LIN {X 0,Y 178.694,Z 336.057,A -85,B 0,C 180,E1 -23455.237,E2 -23455.237} C_VEL
LIN {X 0,Y 177.657,Z 345.122,A -85,B 0,C 180,E1 -23457.721,E2 -23457.721} C_VEL
LIN {X 0,Y 176.562,Z 350.916,A -85,B 0,C 180,E1 -23459.502,E2 -23459.502} C_VEL
LIN {X 0,Y 173.307,Z 359.118,A -85,B 0,C 180,E1 -23462.202,E2 -23462.202} C_VEL
LIN {X 0,Y 169.92,Z 367.179,A -85,B 0,C 180,E1 -23465.569,E2 -23465.569} C_VEL
LIN {X 0,Y 167.647,Z 372.655,A -85,B 0,C 180,E1 -23468.481,E2 -23468.481} C_VEL
LIN {X 0,Y 164.982,Z 378.808,A -85,B 0,C 180,E1 -23472.651,E2 -23472.651} C_VEL
LIN {X 0,Y 163.397,Z 382.822,A -85,B 0,C 180,E1 -23476.316,E2 -23476.316} C_VEL
LIN {X 0,Y 162.479,Z 385.804,A -85,B 0,C 180,E1 -23480.037,E2 -23480.037} C_VEL
LIN {X 0,Y 162.174,Z 387.231,A -85,B 0,C 180,E1 -23482.53,E2 -23482.53} C_VEL
LIN {X 0,Y 162.092,Z 388.497,A -85,B 0,C 180,E1 -23485.741,E2 -23485.741} C_VEL
LIN {X 0,Y 162.298,Z 389.115,A -85,B 0,C 180,E1 -23490,E2 -23490} C_VEL
LIN {X 0,Y 162.074,Z 388.506,A -85,B 0,C 180,E1 -23494.173,E2 -23494.173} C_VEL
LIN {X 0,Y 162.172,Z 387.205,A -85,B 0,C 180,E1 -23497.471,E2 -23497.471} C_VEL
LIN {X 0,Y 162.476,Z 385.767,A -85,B 0,C 180,E1 -23499.964,E2 -23499.964} C_VEL
LIN {X 0,Y 163.397,Z 382.767,A -85,B 0,C 180,E1 -23503.684,E2 -23503.684} C_VEL
LIN {X 0,Y 164.978,Z 378.732,A -85,B 0,C 180,E1 -23507.35,E2 -23507.35} C_VEL
LIN {X 0,Y 167.639,Z 372.55,A -85,B 0,C 180,E1 -23511.521,E2 -23511.521} C_VEL
LIN {X 0,Y 170.317,Z 366.243,A -85,B 0,C 180,E1 -23514.795,E2 -23514.795} C_VEL
LIN {X 0,Y 173.896,Z 357.578,A -85,B 0,C 180,E1 -23518.302,E2 -23518.302} C_VEL
LIN {X 0,Y 174.762,Z 353.72,A -85,B 0,C 180,E1 -23519.737,E2 -23519.737} C_VEL
LIN {X 0,Y 174.495,Z 349.857,A -85,B 0,C 180,E1 -23521.217,E2 -23521.217} C_VEL
LIN {X 0,Y 172.381,Z 339.088,A -85,B 0,C 180,E1 -23525.119,E2 -23525.119} C_VEL
LIN {X 0,Y 172.396,Z 336.052,A -85,B 0,C 180,E1 -23526.015,E2 -23526.015} C_VEL
LIN {X 0,Y 172.819,Z 325.215,A -85,B 0,C 180,E1 -23528.794,E2 -23528.794} C_VEL
LIN {X 0,Y 172.362,Z 314.414,A -85,B 0,C 180,E1 -23531.293,E2 -23531.293} C_VEL
LIN {X 0,Y 171.168,Z 305.853,A -85,B 0,C 180,E1 -23533.214,E2 -23533.214} C_VEL
LIN {X 0,Y 169.717,Z 301.249,A -85,B 0,C 180,E1 -23534.412,E2 -23534.412} C_VEL
LIN {X 0,Y 166.792,Z 294.609,A -85,B 0,C 180,E1 -23536.361,E2 -23536.361} C_VEL
LIN {X 0,Y 164.788,Z 290.322,A -85,B 0,C 180,E1 -23537.639,E2 -23537.639} C_VEL
LIN {X 0,Y 162.711,Z 286.562,A -85,B 0,C 180,E1 -23538.89,E2 -23538.89} C_VEL
LIN {X 0,Y 161.91,Z 284.961,A -85,B 0,C 180,E1 -23539.375,E2 -23539.375} C_VEL
LIN {X 0,Y 159.811,Z 281.715,A -85,B 0,C 180,E1 -23540.586,E2 -23540.586} C_VEL
LIN {X 0,Y 159.083,Z 279.423,A -85,B 0,C 180,E1 -23541.187,E2 -23541.187} C_VEL
LIN {X 0,Y 158.518,Z 275.963,A -85,B 0,C 180,E1 -23547.393,E2 -23547.393} C_VEL
LIN {X 0,Y 158.079,Z 272.941,A -85,B 0,C 180,E1 -23553.603,E2 -23553.603} C_VEL
LIN {X 0,Y 157.67,Z 270.525,A -85,B 0,C 180,E1 -23559.401,E2 -23559.401} C_VEL
LIN {X 0,Y 157.456,Z 268.872,A -85,B 0,C 180,E1 -23564.466,E2 -23564.466} C_VEL
LIN {X 0,Y 157.692,Z 268.842,A -85,B 0,C 180,E1 -23569.731,E2 -23569.731} C_VEL
LIN {X 0,Y 157.769,Z 268.832,A -85,B 0,C 180,E1 -23572.32,E2 -23572.32} C_VEL
LIN {X 0,Y 157.974,Z 268.806,A -85,B 0,C 180,E1 -23577.45,E2 -23577.45} C_VEL
LIN {X 0,Y 158.242,Z 268.772,A -85,B 0,C 180,E1 -23580,E2 -23580} C_VEL
LIN {X 0,Y 157.767,Z 268.833,A -85,B 0,C 180,E1 -23587.68,E2 -23587.68} C_VEL
LIN {X 0,Y 157.636,Z 268.847,A -85,B 0,C 180,E1 -23591.229,E2 -23591.229} C_VEL
LIN {X 0,Y 157.425,Z 268.874,A -85,B 0,C 180,E1 -23595.537,E2 -23595.537} C_VEL
LIN {X 0,Y 157.359,Z 268.881,A -85,B 0,C 180,E1 -23600.935,E2 -23600.935} C_VEL
LIN {X 0,Y 157.312,Z 268.888,A -85,B 0,C 180,E1 -23606.681,E2 -23606.681} C_VEL
LIN {X 0,Y 157.27,Z 268.895,A -85,B 0,C 180,E1 -23612.429,E2 -23612.429} C_VEL
LIN {X 0,Y 157.244,Z 268.897,A -85,B 0,C 180,E1 -23617.473,E2 -23617.473} C_VEL
LIN {X 0,Y 157.215,Z 268.901,A -85,B 0,C 180,E1 -23618.189,E2 -23618.189} C_VEL
LIN {X 0,Y 158.173,Z 271.614,A -85,B 0,C 180,E1 -23618.959,E2 -23618.959} C_VEL
LIN {X 0,Y 160.167,Z 273.789,A -85,B 0,C 180,E1 -23620.092,E2 -23620.092} C_VEL
LIN {X 0,Y 162.728,Z 277.922,A -85,B 0,C 180,E1 -23621.711,E2 -23621.711} C_VEL
LIN {X 0,Y 163.851,Z 279.647,A -85,B 0,C 180,E1 -23622.394,E2 -23622.394} C_VEL
LIN {X 0,Y 167.352,Z 285.536,A -85,B 0,C 180,E1 -23624.619,E2 -23624.619} C_VEL
LIN {X 0,Y 171.406,Z 294.402,A -85,B 0,C 180,E1 -23627.565,E2 -23627.565} C_VEL
LIN {X 0,Y 174.028,Z 302.719,A -85,B 0,C 180,E1 -23630.113,E2 -23630.113} C_VEL
LIN {X 0,Y 175.916,Z 312.518,A -85,B 0,C 180,E1 -23633.037,E2 -23633.037} C_VEL
LIN {X 0,Y 176.6,Z 320.843,A -85,B 0,C 180,E1 -23635.599,E2 -23635.599} C_VEL
LIN {X 0,Y 176.522,Z 323.692,A -85,B 0,C 180,E1 -23636.477,E2 -23636.477} C_VEL
LIN {X 0,Y 173.339,Z 332.499,A -85,B 0,C 180,E1 -23638.872,E2 -23638.872} C_VEL
LIN {X 0,Y 169.236,Z 342.093,A -85,B 0,C 180,E1 -23642.148,E2 -23642.148} C_VEL
LIN {X 0,Y 165.684,Z 349.73,A -85,B 0,C 180,E1 -23645.57,E2 -23645.57} C_VEL
LIN {X 0,Y 162.142,Z 356.74,A -85,B 0,C 180,E1 -23649.71,E2 -23649.71} C_VEL
LIN {X 0,Y 159.687,Z 361.404,A -85,B 0,C 180,E1 -23653.377,E2 -23653.377} C_VEL
LIN {X 0,Y 157.888,Z 364.961,A -85,B 0,C 180,E1 -23657.14,E2 -23657.14} C_VEL
LIN {X 0,Y 156.754,Z 367.275,A -85,B 0,C 180,E1 -23660.527,E2 -23660.527} C_VEL
LIN {X 0,Y 155.826,Z 369.151,A -85,B 0,C 180,E1 -23664.824,E2 -23664.824} C_VEL
LIN {X 0,Y 155.406,Z 369.98,A -85,B 0,C 180,E1 -23670,E2 -23670} C_VEL
LIN {X 0,Y 155.513,Z 369.784,A -85,B 0,C 180,E1 -23672.59,E2 -23672.59} C_VEL
LIN {X 0,Y 155.814,Z 369.201,A -85,B 0,C 180,E1 -23675.175,E2 -23675.175} C_VEL
LIN {X 0,Y 156.942,Z 366.896,A -85,B 0,C 180,E1 -23680.318,E2 -23680.318} C_VEL
LIN {X 0,Y 158.396,Z 364.048,A -85,B 0,C 180,E1 -23684.124,E2 -23684.124} C_VEL
LIN {X 0,Y 160.389,Z 360.182,A -85,B 0,C 180,E1 -23687.862,E2 -23687.862} C_VEL
LIN {X 0,Y 162.993,Z 355.185,A -85,B 0,C 180,E1 -23691.5,E2 -23691.5} C_VEL
LIN {X 0,Y 166.103,Z 348.887,A -85,B 0,C 180,E1 -23695.031,E2 -23695.031} C_VEL
LIN {X 0,Y 169.836,Z 340.996,A -85,B 0,C 180,E1 -23698.417,E2 -23698.417} C_VEL
LIN {X 0,Y 173.294,Z 332.948,A -85,B 0,C 180,E1 -23701.137,E2 -23701.137} C_VEL
LIN {X 0,Y 176.772,Z 323.142,A -85,B 0,C 180,E1 -23703.821,E2 -23703.821} C_VEL
LIN {X 0,Y 176.286,Z 315.562,A -85,B 0,C 180,E1 -23706.21,E2 -23706.21} C_VEL
LIN {X 0,Y 174.842,Z 306.158,A -85,B 0,C 180,E1 -23709.041,E2 -23709.041} C_VEL
LIN {X 0,Y 172.954,Z 298.802,A -85,B 0,C 180,E1 -23711.256,E2 -23711.256} C_VEL
LIN {X 0,Y 169.65,Z 290.247,A -85,B 0,C 180,E1 -23713.981,E2 -23713.981} C_VEL
LIN {X 0,Y 165.677,Z 282.509,A -85,B 0,C 180,E1 -23716.682,E2 -23716.682} C_VEL
LIN {X 0,Y 162.745,Z 277.931,A -85,B 0,C 180,E1 -23718.501,E2 -23718.501} C_VEL
LIN {X 0,Y 160.785,Z 274.801,A -85,B 0,C 180,E1 -23719.739,E2 -23719.739} C_VEL
LIN {X 0,Y 160.185,Z 273.812,A -85,B 0,C 180,E1 -23720.126,E2 -23720.126} C_VEL
LIN {X 0,Y 158.103,Z 271.534,A -85,B 0,C 180,E1 -23721.317,E2 -23721.317} C_VEL
LIN {X 0,Y 157.207,Z 268.903,A -85,B 0,C 180,E1 -23722.045,E2 -23722.045} C_VEL
LIN {X 0,Y 157.279,Z 268.894,A -85,B 0,C 180,E1 -23724.486,E2 -23724.486} C_VEL
LIN {X 0,Y 157.284,Z 268.89,A -85,B 0,C 180,E1 -23728.102,E2 -23728.102} C_VEL
LIN {X 0,Y 157.31,Z 268.889,A -85,B 0,C 180,E1 -23733.464,E2 -23733.464} C_VEL
LIN {X 0,Y 157.378,Z 268.882,A -85,B 0,C 180,E1 -23739.684,E2 -23739.684} C_VEL
LIN {X 0,Y 157.426,Z 268.873,A -85,B 0,C 180,E1 -23744.463,E2 -23744.463} C_VEL
LIN {X 0,Y 157.748,Z 268.831,A -85,B 0,C 180,E1 -23749.734,E2 -23749.734} C_VEL
LIN {X 0,Y 157.82,Z 268.822,A -85,B 0,C 180,E1 -23752.322,E2 -23752.322} C_VEL
LIN {X 0,Y 158.241,Z 268.769,A -85,B 0,C 180,E1 -23760,E2 -23760} C_VEL
LIN {X 0,Y 157.714,Z 268.841,A -85,B 0,C 180,E1 -23765.113,E2 -23765.113} C_VEL
LIN {X 0,Y 157.768,Z 268.833,A -85,B 0,C 180,E1 -23767.68,E2 -23767.68} C_VEL
LIN {X 0,Y 157.659,Z 268.847,A -85,B 0,C 180,E1 -23771.275,E2 -23771.275} C_VEL
LIN {X 0,Y 157.443,Z 268.869,A -85,B 0,C 180,E1 -23775.535,E2 -23775.535} C_VEL
LIN {X 0,Y 157.696,Z 270.702,A -85,B 0,C 180,E1 -23780.887,E2 -23780.887} C_VEL
LIN {X 0,Y 158.056,Z 273.015,A -85,B 0,C 180,E1 -23786.401,E2 -23786.401} C_VEL
LIN {X 0,Y 158.487,Z 276.059,A -85,B 0,C 180,E1 -23792.59,E2 -23792.59} C_VEL
LIN {X 0,Y 159.068,Z 279.471,A -85,B 0,C 180,E1 -23798.716,E2 -23798.716} C_VEL
LIN {X 0,Y 160.384,Z 282.857,A -85,B 0,C 180,E1 -23799.652,E2 -23799.652} C_VEL
LIN {X 0,Y 162.485,Z 285.847,A -85,B 0,C 180,E1 -23800.826,E2 -23800.826} C_VEL
LIN {X 0,Y 164.332,Z 289.647,A -85,B 0,C 180,E1 -23801.994,E2 -23801.994} C_VEL
LIN {X 0,Y 165.621,Z 292.033,A -85,B 0,C 180,E1 -23802.762,E2 -23802.762} C_VEL
LIN {X 0,Y 169.159,Z 299.71,A -85,B 0,C 180,E1 -23805.066,E2 -23805.066} C_VEL
LIN {X 0,Y 171.197,Z 305.8,A -85,B 0,C 180,E1 -23806.69,E2 -23806.69} C_VEL
LIN {X 0,Y 172.473,Z 314.952,A -85,B 0,C 180,E1 -23808.755,E2 -23808.755} C_VEL
LIN {X 0,Y 172.901,Z 325.446,A -85,B 0,C 180,E1 -23811.2,E2 -23811.2} C_VEL
LIN {X 0,Y 172.449,Z 336.06,A -85,B 0,C 180,E1 -23813.921,E2 -23813.921} C_VEL
LIN {X 0,Y 171.405,Z 344.677,A -85,B 0,C 180,E1 -23816.391,E2 -23816.391} C_VEL
LIN {X 0,Y 169.797,Z 352.288,A -85,B 0,C 180,E1 -23818.843,E2 -23818.843} C_VEL
LIN {X 0,Y 165.739,Z 361.567,A -85,B 0,C 180,E1 -23822.196,E2 -23822.196} C_VEL
LIN {X 0,Y 162.419,Z 369.198,A -85,B 0,C 180,E1 -23825.816,E2 -23825.816} C_VEL
LIN {X 0,Y 159.707,Z 375.066,A -85,B 0,C 180,E1 -23829.388,E2 -23829.388} C_VEL
LIN {X 0,Y 157.535,Z 379.828,A -85,B 0,C 180,E1 -23833.143,E2 -23833.143} C_VEL
LIN {X 0,Y 156.082,Z 383.483,A -85,B 0,C 180,E1 -23836.989,E2 -23836.989} C_VEL
LIN {X 0,Y 155.464,Z 385.375,A -85,B 0,C 180,E1 -23839.582,E2 -23839.582} C_VEL
LIN {X 0,Y 155.011,Z 387.829,A -85,B 0,C 180,E1 -23844.798,E2 -23844.798} C_VEL
LIN {X 0,Y 155.026,Z 388.459,A -85,B 0,C 180,E1 -23847.402,E2 -23847.402} C_VEL
LIN {X 0,Y 155.214,Z 388.689,A -85,B 0,C 180,E1 -23850,E2 -23850} C_VEL
LIN {X 0,Y 155.002,Z 388.164,A -85,B 0,C 180,E1 -23854.045,E2 -23854.045} C_VEL
LIN {X 0,Y 155.111,Z 386.776,A -85,B 0,C 180,E1 -23857.813,E2 -23857.813} C_VEL
LIN {X 0,Y 155.462,Z 385.337,A -85,B 0,C 180,E1 -23860.418,E2 -23860.418} C_VEL
LIN {X 0,Y 156.468,Z 382.336,A -85,B 0,C 180,E1 -23864.303,E2 -23864.303} C_VEL
LIN {X 0,Y 158.195,Z 378.302,A -85,B 0,C 180,E1 -23868.119,E2 -23868.119} C_VEL
LIN {X 0,Y 161.045,Z 372.12,A -85,B 0,C 180,E1 -23872.449,E2 -23872.449} C_VEL
LIN {X 0,Y 163.99,Z 365.503,A -85,B 0,C 180,E1 -23875.989,E2 -23875.989} C_VEL
LIN {X 0,Y 167.695,Z 357.031,A -85,B 0,C 180,E1 -23879.501,E2 -23879.501} C_VEL
LIN {X 0,Y 169.785,Z 352.093,A -85,B 0,C 180,E1 -23881.16,E2 -23881.16} C_VEL
LIN {X 0,Y 171.535,Z 343.379,A -85,B 0,C 180,E1 -23883.934,E2 -23883.934} C_VEL
LIN {X 0,Y 172.396,Z 336.052,A -85,B 0,C 180,E1 -23886.015,E2 -23886.015} C_VEL
LIN {X 0,Y 172.137,Z 331.689,A -85,B 0,C 180,E1 -23887.336,E2 -23887.336} C_VEL
LIN {X 0,Y 170.969,Z 327.609,A -85,B 0,C 180,E1 -23888.729,E2 -23888.729} C_VEL
LIN {X 0,Y 167.747,Z 319.532,A -85,B 0,C 180,E1 -23891.534,E2 -23891.534} C_VEL
LIN {X 0,Y 166.552,Z 315.06,A -85,B 0,C 180,E1 -23892.841,E2 -23892.841} C_VEL
LIN {X 0,Y 166.322,Z 313.452,A -85,B 0,C 180,E1 -23893.241,E2 -23893.241} C_VEL
LIN {X 0,Y 165.249,Z 307.101,A -85,B 0,C 180,E1 -23894.848,E2 -23894.848} C_VEL
LIN {X 0,Y 161.779,Z 298.409,A -85,B 0,C 180,E1 -23897.606,E2 -23897.606} C_VEL
LIN {X 0,Y 160.213,Z 294.941,A -85,B 0,C 180,E1 -23898.744,E2 -23898.744} C_VEL
LIN {X 0,Y 157.631,Z 289.802,A -85,B 0,C 180,E1 -23900.555,E2 -23900.555} C_VEL
LIN {X 0,Y 155.501,Z 285.739,A -85,B 0,C 180,E1 -23902.049,E2 -23902.049} C_VEL
LIN {X 0,Y 154.729,Z 284.47,A -85,B 0,C 180,E1 -23902.555,E2 -23902.555} C_VEL
LIN {X 0,Y 152.517,Z 281.225,A -85,B 0,C 180,E1 -23904.019,E2 -23904.019} C_VEL
LIN {X 0,Y 151.752,Z 278.759,A -85,B 0,C 180,E1 -23904.728,E2 -23904.728} C_VEL
LIN {X 0,Y 151.369,Z 276.46,A -85,B 0,C 180,E1 -23909.288,E2 -23909.288} C_VEL
LIN {X 0,Y 151.205,Z 275.058,A -85,B 0,C 180,E1 -23912.303,E2 -23912.303} C_VEL
LIN {X 0,Y 150.771,Z 272.37,A -85,B 0,C 180,E1 -23918.794,E2 -23918.794} C_VEL
LIN {X 0,Y 150.54,Z 270.645,A -85,B 0,C 180,E1 -23923.733,E2 -23923.733} C_VEL
LIN {X 0,Y 150.445,Z 269.8,A -85,B 0,C 180,E1 -23926.493,E2 -23926.493} C_VEL
LIN {X 0,Y 150.626,Z 269.724,A -85,B 0,C 180,E1 -23929.244,E2 -23929.244} C_VEL
LIN {X 0,Y 150.707,Z 269.713,A -85,B 0,C 180,E1 -23931.958,E2 -23931.958} C_VEL
LIN {X 0,Y 151.204,Z 269.649,A -85,B 0,C 180,E1 -23940,E2 -23940} C_VEL
LIN {X 0,Y 150.705,Z 269.712,A -85,B 0,C 180,E1 -23948.042,E2 -23948.042} C_VEL
LIN {X 0,Y 150.578,Z 269.726,A -85,B 0,C 180,E1 -23951.433,E2 -23951.433} C_VEL
LIN {X 0,Y 150.333,Z 269.759,A -85,B 0,C 180,E1 -23956.29,E2 -23956.29} C_VEL
LIN {X 0,Y 150.342,Z 269.755,A -85,B 0,C 180,E1 -23960.78,E2 -23960.78} C_VEL
LIN {X 0,Y 150.241,Z 269.771,A -85,B 0,C 180,E1 -23967.277,E2 -23967.277} C_VEL
LIN {X 0,Y 150.211,Z 269.773,A -85,B 0,C 180,E1 -23972.628,E2 -23972.628} C_VEL
LIN {X 0,Y 150.188,Z 269.775,A -85,B 0,C 180,E1 -23974.67,E2 -23974.67} C_VEL
LIN {X 0,Y 151.132,Z 272.438,A -85,B 0,C 180,E1 -23975.541,E2 -23975.541} C_VEL
LIN {X 0,Y 153.125,Z 274.667,A -85,B 0,C 180,E1 -23976.874,E2 -23976.874} C_VEL
LIN {X 0,Y 153.818,Z 275.484,A -85,B 0,C 180,E1 -23977.344,E2 -23977.344} C_VEL
LIN {X 0,Y 155.642,Z 278.625,A -85,B 0,C 180,E1 -23978.697,E2 -23978.697} C_VEL
LIN {X 0,Y 157.036,Z 280.466,A -85,B 0,C 180,E1 -23979.624,E2 -23979.624} C_VEL
LIN {X 0,Y 160.948,Z 287.028,A -85,B 0,C 180,E1 -23982.427,E2 -23982.427} C_VEL
LIN {X 0,Y 164.358,Z 293.877,A -85,B 0,C 180,E1 -23985.052,E2 -23985.052} C_VEL
LIN {X 0,Y 166.932,Z 300.819,A -85,B 0,C 180,E1 -23987.459,E2 -23987.459} C_VEL
LIN {X 0,Y 168.746,Z 307.844,A -85,B 0,C 180,E1 -23989.763,E2 -23989.763} C_VEL
LIN {X 0,Y 170.042,Z 316.864,A -85,B 0,C 180,E1 -23992.67,E2 -23992.67} C_VEL
LIN {X 0,Y 170.378,Z 324.858,A -85,B 0,C 180,E1 -23995.347,E2 -23995.347} C_VEL
LIN {X 0,Y 166.591,Z 334.695,A -85,B 0,C 180,E1 -23998.173,E2 -23998.173} C_VEL
LIN {X 0,Y 163.016,Z 342.522,A -85,B 0,C 180,E1 -24000.986,E2 -24000.986} C_VEL
LIN {X 0,Y 159.26,Z 350.158,A -85,B 0,C 180,E1 -24004.516,E2 -24004.516} C_VEL
LIN {X 0,Y 155.519,Z 357.169,A -85,B 0,C 180,E1 -24008.806,E2 -24008.806} C_VEL
LIN {X 0,Y 152.912,Z 361.832,A -85,B 0,C 180,E1 -24012.617,E2 -24012.617} C_VEL
LIN {X 0,Y 150.973,Z 365.389,A -85,B 0,C 180,E1 -24016.54,E2 -24016.54} C_VEL
LIN {X 0,Y 149.684,Z 367.872,A -85,B 0,C 180,E1 -24020.402,E2 -24020.402} C_VEL
LIN {X 0,Y 148.776,Z 369.578,A -85,B 0,C 180,E1 -24024.578,E2 -24024.578} C_VEL
LIN {X 0,Y 148.347,Z 370.405,A -85,B 0,C 180,E1 -24030,E2 -24030} C_VEL
LIN {X 0,Y 148.439,Z 370.21,A -85,B 0,C 180,E1 -24032.713,E2 -24032.713} C_VEL
LIN {X 0,Y 148.763,Z 369.627,A -85,B 0,C 180,E1 -24035.421,E2 -24035.421} C_VEL
LIN {X 0,Y 149.982,Z 367.322,A -85,B 0,C 180,E1 -24040.803,E2 -24040.803} C_VEL
LIN {X 0,Y 151.534,Z 364.474,A -85,B 0,C 180,E1 -24044.778,E2 -24044.778} C_VEL
LIN {X 0,Y 153.649,Z 360.608,A -85,B 0,C 180,E1 -24048.674,E2 -24048.674} C_VEL
LIN {X 0,Y 156.419,Z 355.61,A -85,B 0,C 180,E1 -24052.452,E2 -24052.452} C_VEL
LIN {X 0,Y 159.703,Z 349.312,A -85,B 0,C 180,E1 -24056.108,E2 -24056.108} C_VEL
LIN {X 0,Y 163.643,Z 341.42,A -85,B 0,C 180,E1 -24059.597,E2 -24059.597} C_VEL
LIN {X 0,Y 167.265,Z 333.372,A -85,B 0,C 180,E1 -24062.392,E2 -24062.392} C_VEL
LIN {X 0,Y 170.487,Z 324.68,A -85,B 0,C 180,E1 -24064.87,E2 -24064.87} C_VEL
LIN {X 0,Y 170.066,Z 316.091,A -85,B 0,C 180,E1 -24067.741,E2 -24067.741} C_VEL
LIN {X 0,Y 168.502,Z 306.306,A -85,B 0,C 180,E1 -24070.9,E2 -24070.9} C_VEL
LIN {X 0,Y 165.814,Z 297.331,A -85,B 0,C 180,E1 -24073.9,E2 -24073.9} C_VEL
LIN {X 0,Y 162.05,Z 288.967,A -85,B 0,C 180,E1 -24077.001,E2 -24077.001} C_VEL
LIN {X 0,Y 158.675,Z 283.229,A -85,B 0,C 180,E1 -24079.418,E2 -24079.418} C_VEL
LIN {X 0,Y 156.462,Z 279.471,A -85,B 0,C 180,E1 -24081.034,E2 -24081.034} C_VEL
LIN {X 0,Y 154.281,Z 276.557,A -85,B 0,C 180,E1 -24082.509,E2 -24082.509} C_VEL
LIN {X 0,Y 153.407,Z 274.854,A -85,B 0,C 180,E1 -24083.206,E2 -24083.206} C_VEL
LIN {X 0,Y 151.282,Z 272.7,A -85,B 0,C 180,E1 -24084.602,E2 -24084.602} C_VEL
LIN {X 0,Y 150.285,Z 270.385,A -85,B 0,C 180,E1 -24085.457,E2 -24085.457} C_VEL
LIN {X 0,Y 150.195,Z 269.774,A -85,B 0,C 180,E1 -24085.637,E2 -24085.637} C_VEL
LIN {X 0,Y 150.192,Z 269.773,A -85,B 0,C 180,E1 -24089.02,E2 -24089.02} C_VEL
LIN {X 0,Y 150.239,Z 269.771,A -85,B 0,C 180,E1 -24092.722,E2 -24092.722} C_VEL
LIN {X 0,Y 150.34,Z 269.756,A -85,B 0,C 180,E1 -24099.22,E2 -24099.22} C_VEL
LIN {X 0,Y 150.333,Z 269.759,A -85,B 0,C 180,E1 -24103.71,E2 -24103.71} C_VEL
LIN {X 0,Y 150.662,Z 269.713,A -85,B 0,C 180,E1 -24109.246,E2 -24109.246} C_VEL
LIN {X 0,Y 150.756,Z 269.703,A -85,B 0,C 180,E1 -24111.96,E2 -24111.96} C_VEL
LIN {X 0,Y 151.203,Z 269.646,A -85,B 0,C 180,E1 -24120,E2 -24120} C_VEL
LIN {X 0,Y 150.705,Z 269.714,A -85,B 0,C 180,E1 -24128.042,E2 -24128.042} C_VEL
LIN {X 0,Y 150.591,Z 269.726,A -85,B 0,C 180,E1 -24131.461,E2 -24131.461} C_VEL
LIN {X 0,Y 150.448,Z 269.87,A -85,B 0,C 180,E1 -24133.507,E2 -24133.507} C_VEL
LIN {X 0,Y 150.684,Z 271.655,A -85,B 0,C 180,E1 -24139.055,E2 -24139.055} C_VEL
LIN {X 0,Y 150.952,Z 273.87,A -85,B 0,C 180,E1 -24144.773,E2 -24144.773} C_VEL
LIN {X 0,Y 151.183,Z 275.265,A -85,B 0,C 180,E1 -24147.964,E2 -24147.964} C_VEL
LIN {X 0,Y 151.585,Z 278.099,A -85,B 0,C 180,E1 -24153.804,E2 -24153.804} C_VEL
LIN {X 0,Y 151.745,Z 278.823,A -85,B 0,C 180,E1 -24155.172,E2 -24155.172} C_VEL
LIN {X 0,Y 152.756,Z 281.769,A -85,B 0,C 180,E1 -24156.018,E2 -24156.018} C_VEL
LIN {X 0,Y 155.488,Z 285.652,A -85,B 0,C 180,E1 -24157.796,E2 -24157.796} C_VEL
LIN {X 0,Y 157.33,Z 289.336,A -85,B 0,C 180,E1 -24159.122,E2 -24159.122} C_VEL
LIN {X 0,Y 158.516,Z 291.379,A -85,B 0,C 180,E1 -24159.903,E2 -24159.903} C_VEL
LIN {X 0,Y 161.197,Z 296.995,A -85,B 0,C 180,E1 -24161.831,E2 -24161.831} C_VEL
LIN {X 0,Y 164.503,Z 304.814,A -85,B 0,C 180,E1 -24164.369,E2 -24164.369} C_VEL
LIN {X 0,Y 166.074,Z 310.645,A -85,B 0,C 180,E1 -24166.006,E2 -24166.006} C_VEL
LIN {X 0,Y 166.793,Z 320.116,A -85,B 0,C 180,E1 -24168.292,E2 -24168.292} C_VEL
LIN {X 0,Y 166.747,Z 329.849,A -85,B 0,C 180,E1 -24170.786,E2 -24170.786} C_VEL
LIN {X 0,Y 165.899,Z 339.888,A -85,B 0,C 180,E1 -24173.624,E2 -24173.624} C_VEL
LIN {X 0,Y 164.496,Z 348.209,A -85,B 0,C 180,E1 -24176.261,E2 -24176.261} C_VEL
LIN {X 0,Y 163.019,Z 353.542,A -85,B 0,C 180,E1 -24178.122,E2 -24178.122} C_VEL
LIN {X 0,Y 158.812,Z 362.507,A -85,B 0,C 180,E1 -24181.594,E2 -24181.594} C_VEL
LIN {X 0,Y 155.567,Z 369.55,A -85,B 0,C 180,E1 -24185.172,E2 -24185.172} C_VEL
LIN {X 0,Y 153.026,Z 374.636,A -85,B 0,C 180,E1 -24188.444,E2 -24188.444} C_VEL
LIN {X 0,Y 150.71,Z 379.399,A -85,B 0,C 180,E1 -24192.356,E2 -24192.356} C_VEL
LIN {X 0,Y 149.123,Z 383.053,A -85,B 0,C 180,E1 -24196.371,E2 -24196.371} C_VEL
LIN {X 0,Y 148.469,Z 384.947,A -85,B 0,C 180,E1 -24199.086,E2 -24199.086} C_VEL
LIN {X 0,Y 147.929,Z 387.401,A -85,B 0,C 180,E1 -24204.548,E2 -24204.548} C_VEL
LIN {X 0,Y 147.933,Z 388.031,A -85,B 0,C 180,E1 -24207.277,E2 -24207.277} C_VEL
LIN {X 0,Y 148.13,Z 388.262,A -85,B 0,C 180,E1 -24210,E2 -24210} C_VEL
LIN {X 0,Y 147.94,Z 387.793,A -85,B 0,C 180,E1 -24213.95,E2 -24213.95} C_VEL
LIN {X 0,Y 148.044,Z 386.346,A -85,B 0,C 180,E1 -24218.188,E2 -24218.188} C_VEL
LIN {X 0,Y 148.467,Z 384.907,A -85,B 0,C 180,E1 -24220.915,E2 -24220.915} C_VEL
LIN {X 0,Y 149.566,Z 381.906,A -85,B 0,C 180,E1 -24224.978,E2 -24224.978} C_VEL
LIN {X 0,Y 151.416,Z 377.87,A -85,B 0,C 180,E1 -24228.96,E2 -24228.96} C_VEL
LIN {X 0,Y 154.499,Z 371.69,A -85,B 0,C 180,E1 -24233.456,E2 -24233.456} C_VEL
LIN {X 0,Y 157.664,Z 364.945,A -85,B 0,C 180,E1 -24237.188,E2 -24237.188} C_VEL
LIN {X 0,Y 161.54,Z 356.6,A -85,B 0,C 180,E1 -24240.744,E2 -24240.744} C_VEL
LIN {X 0,Y 163.566,Z 351.649,A -85,B 0,C 180,E1 -24242.486,E2 -24242.486} C_VEL
LIN {X 0,Y 165.393,Z 342.872,A -85,B 0,C 180,E1 -24245.397,E2 -24245.397} C_VEL
LIN {X 0,Y 166.436,Z 333.537,A -85,B 0,C 180,E1 -24248.139,E2 -24248.139} C_VEL
LIN {X 0,Y 166.816,Z 322.544,A -85,B 0,C 180,E1 -24251.011,E2 -24251.011} C_VEL
LIN {X 0,Y 166.322,Z 313.452,A -85,B 0,C 180,E1 -24253.241,E2 -24253.241} C_VEL
LIN {X 0,Y 165.664,Z 310.424,A -85,B 0,C 180,E1 -24254.069,E2 -24254.069} C_VEL
LIN {X 0,Y 164.464,Z 307.771,A -85,B 0,C 180,E1 -24254.985,E2 -24254.985} C_VEL
LIN {X 0,Y 161.161,Z 303.358,A -85,B 0,C 180,E1 -24256.995,E2 -24256.995} C_VEL
LIN {X 0,Y 153.729,Z 295.243,A -85,B 0,C 180,E1 -24261.424,E2 -24261.424} C_VEL
LIN {X 0,Y 151.603,Z 290.966,A -85,B 0,C 180,E1 -24263.148,E2 -24263.148} C_VEL
LIN {X 0,Y 148.668,Z 285.889,A -85,B 0,C 180,E1 -24265.439,E2 -24265.439} C_VEL
LIN {X 0,Y 147.872,Z 284.147,A -85,B 0,C 180,E1 -24266.123,E2 -24266.123} C_VEL
LIN {X 0,Y 145.349,Z 280.732,A -85,B 0,C 180,E1 -24268.072,E2 -24268.072} C_VEL
LIN {X 0,Y 144.432,Z 278.009,A -85,B 0,C 180,E1 -24269.072,E2 -24269.072} C_VEL
LIN {X 0,Y 144.083,Z 275.856,A -85,B 0,C 180,E1 -24273.96,E2 -24273.96} C_VEL
LIN {X 0,Y 143.776,Z 273.541,A -85,B 0,C 180,E1 -24279.991,E2 -24279.991} C_VEL
LIN {X 0,Y 143.554,Z 271.697,A -85,B 0,C 180,E1 -24285.831,E2 -24285.831} C_VEL
LIN {X 0,Y 143.597,Z 270.883,A -85,B 0,C 180,E1 -24288.71,E2 -24288.71} C_VEL
LIN {X 0,Y 143.63,Z 270.596,A -85,B 0,C 180,E1 -24291.559,E2 -24291.559} C_VEL
LIN {X 0,Y 144.164,Z 270.526,A -85,B 0,C 180,E1 -24300,E2 -24300} C_VEL
LIN {X 0,Y 143.627,Z 270.592,A -85,B 0,C 180,E1 -24308.442,E2 -24308.442} C_VEL
LIN {X 0,Y 143.504,Z 270.606,A -85,B 0,C 180,E1 -24311.621,E2 -24311.621} C_VEL
LIN {X 0,Y 143.272,Z 270.636,A -85,B 0,C 180,E1 -24317.117,E2 -24317.117} C_VEL
LIN {X 0,Y 143.269,Z 270.637,A -85,B 0,C 180,E1 -24321.244,E2 -24321.244} C_VEL
LIN {X 0,Y 143.185,Z 270.648,A -85,B 0,C 180,E1 -24327.931,E2 -24327.931} C_VEL
LIN {X 0,Y 143.168,Z 270.851,A -85,B 0,C 180,E1 -24330.413,E2 -24330.413} C_VEL
LIN {X 0,Y 144.077,Z 273.378,A -85,B 0,C 180,E1 -24331.422,E2 -24331.422} C_VEL
LIN {X 0,Y 146.25,Z 275.679,A -85,B 0,C 180,E1 -24333.159,E2 -24333.159} C_VEL
LIN {X 0,Y 147.004,Z 276.3,A -85,B 0,C 180,E1 -24333.725,E2 -24333.725} C_VEL
LIN {X 0,Y 148.731,Z 279.486,A -85,B 0,C 180,E1 -24335.266,E2 -24335.266} C_VEL
LIN {X 0,Y 150.329,Z 281.442,A -85,B 0,C 180,E1 -24336.485,E2 -24336.485} C_VEL
LIN {X 0,Y 154.983,Z 289.096,A -85,B 0,C 180,E1 -24340.256,E2 -24340.256} C_VEL
LIN {X 0,Y 157.922,Z 294.771,A -85,B 0,C 180,E1 -24342.74,E2 -24342.74} C_VEL
LIN {X 0,Y 160.864,Z 302.141,A -85,B 0,C 180,E1 -24345.65,E2 -24345.65} C_VEL
LIN {X 0,Y 163.002,Z 310.677,A -85,B 0,C 180,E1 -24348.694,E2 -24348.694} C_VEL
LIN {X 0,Y 164.026,Z 319.692,A -85,B 0,C 180,E1 -24351.815,E2 -24351.815} C_VEL
LIN {X 0,Y 164.195,Z 325.419,A -85,B 0,C 180,E1 -24353.878,E2 -24353.878} C_VEL
LIN {X 0,Y 163.868,Z 327.319,A -85,B 0,C 180,E1 -24354.485,E2 -24354.485} C_VEL
LIN {X 0,Y 159.848,Z 336.804,A -85,B 0,C 180,E1 -24357.411,E2 -24357.411} C_VEL
LIN {X 0,Y 155.479,Z 345.669,A -85,B 0,C 180,E1 -24360.926,E2 -24360.926} C_VEL
LIN {X 0,Y 151.707,Z 352.794,A -85,B 0,C 180,E1 -24364.626,E2 -24364.626} C_VEL
LIN {X 0,Y 148.944,Z 357.596,A -85,B 0,C 180,E1 -24367.822,E2 -24367.822} C_VEL
LIN {X 0,Y 146.175,Z 362.259,A -85,B 0,C 180,E1 -24371.789,E2 -24371.789} C_VEL
LIN {X 0,Y 144.097,Z 365.817,A -85,B 0,C 180,E1 -24375.885,E2 -24375.885} C_VEL
LIN {X 0,Y 142.563,Z 368.534,A -85,B 0,C 180,E1 -24380.387,E2 -24380.387} C_VEL
LIN {X 0,Y 141.731,Z 370.005,A -85,B 0,C 180,E1 -24384.308,E2 -24384.308} C_VEL
LIN {X 0,Y 141.265,Z 370.832,A -85,B 0,C 180,E1 -24390,E2 -24390} C_VEL
LIN {X 0,Y 141.367,Z 370.637,A -85,B 0,C 180,E1 -24392.849,E2 -24392.849} C_VEL
LIN {X 0,Y 141.717,Z 370.053,A -85,B 0,C 180,E1 -24395.692,E2 -24395.692} C_VEL
LIN {X 0,Y 142.456,Z 368.752,A -85,B 0,C 180,E1 -24399.355,E2 -24399.355} C_VEL
LIN {X 0,Y 144.084,Z 365.945,A -85,B 0,C 180,E1 -24404.116,E2 -24404.116} C_VEL
LIN {X 0,Y 146.142,Z 362.436,A -85,B 0,C 180,E1 -24408.215,E2 -24408.215} C_VEL
LIN {X 0,Y 148.878,Z 357.823,A -85,B 0,C 180,E1 -24412.188,E2 -24412.188} C_VEL
LIN {X 0,Y 152.776,Z 350.866,A -85,B 0,C 180,E1 -24416.648,E2 -24416.648} C_VEL
LIN {X 0,Y 156.809,Z 343.31,A -85,B 0,C 180,E1 -24420.279,E2 -24420.279} C_VEL
LIN {X 0,Y 160.565,Z 335.561,A -85,B 0,C 180,E1 -24423.17,E2 -24423.17} C_VEL
LIN {X 0,Y 164.259,Z 326.324,A -85,B 0,C 180,E1 -24425.961,E2 -24425.961} C_VEL
LIN {X 0,Y 163.974,Z 317.751,A -85,B 0,C 180,E1 -24429.027,E2 -24429.027} C_VEL
LIN {X 0,Y 162.642,Z 308.715,A -85,B 0,C 180,E1 -24432.182,E2 -24432.182} C_VEL
LIN {X 0,Y 160.118,Z 299.983,A -85,B 0,C 180,E1 -24435.389,E2 -24435.389} C_VEL
LIN {X 0,Y 157.391,Z 293.646,A -85,B 0,C 180,E1 -24437.948,E2 -24437.948} C_VEL
LIN {X 0,Y 154.398,Z 288.294,A -85,B 0,C 180,E1 -24440.412,E2 -24440.412} C_VEL
LIN {X 0,Y 152.116,Z 284.438,A -85,B 0,C 180,E1 -24442.284,E2 -24442.284} C_VEL
LIN {X 0,Y 149.715,Z 280.528,A -85,B 0,C 180,E1 -24444.278,E2 -24444.278} C_VEL
LIN {X 0,Y 147.528,Z 277.559,A -85,B 0,C 180,E1 -24446.02,E2 -24446.02} C_VEL
LIN {X 0,Y 146.699,Z 275.938,A -85,B 0,C 180,E1 -24446.801,E2 -24446.801} C_VEL
LIN {X 0,Y 144.423,Z 273.922,A -85,B 0,C 180,E1 -24448.56,E2 -24448.56} C_VEL
LIN {X 0,Y 143.21,Z 271.242,A -85,B 0,C 180,E1 -24449.8,E2 -24449.8} C_VEL
LIN {X 0,Y 143.107,Z 270.66,A -85,B 0,C 180,E1 -24449.979,E2 -24449.979} C_VEL
LIN {X 0,Y 143.151,Z 270.651,A -85,B 0,C 180,E1 -24453.777,E2 -24453.777} C_VEL
LIN {X 0,Y 143.285,Z 270.638,A -85,B 0,C 180,E1 -24459.919,E2 -24459.919} C_VEL
LIN {X 0,Y 143.35,Z 270.623,A -85,B 0,C 180,E1 -24465.81,E2 -24465.81} C_VEL
LIN {X 0,Y 143.595,Z 270.593,A -85,B 0,C 180,E1 -24468.71,E2 -24468.71} C_VEL
LIN {X 0,Y 143.675,Z 270.587,A -85,B 0,C 180,E1 -24471.561,E2 -24471.561} C_VEL
LIN {X 0,Y 144.163,Z 270.522,A -85,B 0,C 180,E1 -24480,E2 -24480} C_VEL
LIN {X 0,Y 143.629,Z 270.593,A -85,B 0,C 180,E1 -24488.441,E2 -24488.441} C_VEL
LIN {X 0,Y 143.589,Z 271.097,A -85,B 0,C 180,E1 -24491.789,E2 -24491.789} C_VEL
LIN {X 0,Y 143.657,Z 272.657,A -85,B 0,C 180,E1 -24497.069,E2 -24497.069} C_VEL
LIN {X 0,Y 143.878,Z 274.315,A -85,B 0,C 180,E1 -24501.86,E2 -24501.86} C_VEL
LIN {X 0,Y 144.067,Z 275.951,A -85,B 0,C 180,E1 -24506.043,E2 -24506.043} C_VEL
LIN {X 0,Y 144.434,Z 278.129,A -85,B 0,C 180,E1 -24510.826,E2 -24510.826} C_VEL
LIN {X 0,Y 145.496,Z 281.128,A -85,B 0,C 180,E1 -24511.892,E2 -24511.892} C_VEL
LIN {X 0,Y 148.083,Z 284.369,A -85,B 0,C 180,E1 -24513.858,E2 -24513.858} C_VEL
LIN {X 0,Y 150.112,Z 288.733,A -85,B 0,C 180,E1 -24515.613,E2 -24515.613} C_VEL
LIN {X 0,Y 151.65,Z 291.015,A -85,B 0,C 180,E1 -24516.735,E2 -24516.735} C_VEL
LIN {X 0,Y 153.826,Z 295.341,A -85,B 0,C 180,E1 -24518.499,E2 -24518.499} C_VEL
LIN {X 0,Y 157.841,Z 304.558,A -85,B 0,C 180,E1 -24521.904,E2 -24521.904} C_VEL
LIN {X 0,Y 159.939,Z 310.65,A -85,B 0,C 180,E1 -24523.96,E2 -24523.96} C_VEL
LIN {X 0,Y 160.716,Z 315.314,A -85,B 0,C 180,E1 -24525.284,E2 -24525.284} C_VEL
LIN {X 0,Y 160.953,Z 325.341,A -85,B 0,C 180,E1 -24527.928,E2 -24527.928} C_VEL
LIN {X 0,Y 160.385,Z 334.664,A -85,B 0,C 180,E1 -24530.552,E2 -24530.552} C_VEL
LIN {X 0,Y 159.009,Z 344.556,A -85,B 0,C 180,E1 -24533.672,E2 -24533.672} C_VEL
LIN {X 0,Y 157.474,Z 351.414,A -85,B 0,C 180,E1 -24536.092,E2 -24536.092} C_VEL
LIN {X 0,Y 155.47,Z 356.34,A -85,B 0,C 180,E1 -24537.917,E2 -24537.917} C_VEL
LIN {X 0,Y 151.265,Z 364.648,A -85,B 0,C 180,E1 -24541.561,E2 -24541.561} C_VEL
LIN {X 0,Y 147.997,Z 371.374,A -85,B 0,C 180,E1 -24545.448,E2 -24545.448} C_VEL
LIN {X 0,Y 144.688,Z 377.522,A -85,B 0,C 180,E1 -24550.123,E2 -24550.123} C_VEL
LIN {X 0,Y 142.667,Z 381.534,A -85,B 0,C 180,E1 -24554.28,E2 -24554.28} C_VEL
LIN {X 0,Y 141.46,Z 384.518,A -85,B 0,C 180,E1 -24558.538,E2 -24558.538} C_VEL
LIN {X 0,Y 140.848,Z 386.973,A -85,B 0,C 180,E1 -24564.273,E2 -24564.273} C_VEL
LIN {X 0,Y 140.864,Z 387.605,A -85,B 0,C 180,E1 -24567.141,E2 -24567.141} C_VEL
LIN {X 0,Y 141.048,Z 387.835,A -85,B 0,C 180,E1 -24570,E2 -24570} C_VEL
LIN {X 0,Y 140.843,Z 387.456,A -85,B 0,C 180,E1 -24573.633,E2 -24573.633} C_VEL
LIN {X 0,Y 141.005,Z 385.917,A -85,B 0,C 180,E1 -24578.6,E2 -24578.6} C_VEL
LIN {X 0,Y 141.459,Z 384.477,A -85,B 0,C 180,E1 -24581.463,E2 -24581.463} C_VEL
LIN {X 0,Y 142.667,Z 381.474,A -85,B 0,C 180,E1 -24585.721,E2 -24585.721} C_VEL
LIN {X 0,Y 144.68,Z 377.439,A -85,B 0,C 180,E1 -24589.879,E2 -24589.879} C_VEL
LIN {X 0,Y 148.002,Z 371.26,A -85,B 0,C 180,E1 -24594.552,E2 -24594.552} C_VEL
LIN {X 0,Y 151.346,Z 364.513,A -85,B 0,C 180,E1 -24598.424,E2 -24598.424} C_VEL
LIN {X 0,Y 155.469,Z 356.169,A -85,B 0,C 180,E1 -24602.085,E2 -24602.085} C_VEL
LIN {X 0,Y 157.431,Z 351.205,A -85,B 0,C 180,E1 -24603.92,E2 -24603.92} C_VEL
LIN {X 0,Y 159.349,Z 342.236,A -85,B 0,C 180,E1 -24607.021,E2 -24607.021} C_VEL
LIN {X 0,Y 160.555,Z 331.742,A -85,B 0,C 180,E1 -24610.215,E2 -24610.215} C_VEL
LIN {X 0,Y 160.916,Z 322.186,A -85,B 0,C 180,E1 -24612.831,E2 -24612.831} C_VEL
LIN {X 0,Y 160.29,Z 312.268,A -85,B 0,C 180,E1 -24615.45,E2 -24615.45} C_VEL
LIN {X 0,Y 157.726,Z 304.369,A -85,B 0,C 180,E1 -24618.058,E2 -24618.058} C_VEL
LIN {X 0,Y 153.729,Z 295.243,A -85,B 0,C 180,E1 -24621.424,E2 -24621.424} C_VEL
LIN {X 0,Y 150.368,Z 291.429,A -85,B 0,C 180,E1 -24623.683,E2 -24623.683} C_VEL
LIN {X 0,Y 143.091,Z 285.873,A -85,B 0,C 180,E1 -24628.739,E2 -24628.739} C_VEL
LIN {X 0,Y 139.957,Z 282.669,A -85,B 0,C 180,E1 -24631.39,E2 -24631.39} C_VEL
LIN {X 0,Y 137.813,Z 279.336,A -85,B 0,C 180,E1 -24633.601,E2 -24633.601} C_VEL
LIN {X 0,Y 137.082,Z 277.128,A -85,B 0,C 180,E1 -24634.572,E2 -24634.572} C_VEL
LIN {X 0,Y 136.902,Z 275.5,A -85,B 0,C 180,E1 -24638.94,E2 -24638.94} C_VEL
LIN {X 0,Y 136.655,Z 273.598,A -85,B 0,C 180,E1 -24645.099,E2 -24645.099} C_VEL
LIN {X 0,Y 136.712,Z 272.758,A -85,B 0,C 180,E1 -24648.134,E2 -24648.134} C_VEL
LIN {X 0,Y 136.642,Z 272.055,A -85,B 0,C 180,E1 -24651.124,E2 -24651.124} C_VEL
LIN {X 0,Y 136.548,Z 271.478,A -85,B 0,C 180,E1 -24654.092,E2 -24654.092} C_VEL
LIN {X 0,Y 137.122,Z 271.403,A -85,B 0,C 180,E1 -24660,E2 -24660} C_VEL
LIN {X 0,Y 136.552,Z 271.472,A -85,B 0,C 180,E1 -24668.882,E2 -24668.882} C_VEL
LIN {X 0,Y 136.418,Z 271.488,A -85,B 0,C 180,E1 -24671.892,E2 -24671.892} C_VEL
LIN {X 0,Y 136.191,Z 271.517,A -85,B 0,C 180,E1 -24678.037,E2 -24678.037} C_VEL
LIN {X 0,Y 136.192,Z 271.52,A -85,B 0,C 180,E1 -24681.739,E2 -24681.739} C_VEL
LIN {X 0,Y 136.077,Z 271.549,A -85,B 0,C 180,E1 -24684.812,E2 -24684.812} C_VEL
LIN {X 0,Y 136.785,Z 273.808,A -85,B 0,C 180,E1 -24685.896,E2 -24685.896} C_VEL
LIN {X 0,Y 138.547,Z 276.025,A -85,B 0,C 180,E1 -24687.793,E2 -24687.793} C_VEL
LIN {X 0,Y 140.277,Z 277.341,A -85,B 0,C 180,E1 -24689.406,E2 -24689.406} C_VEL
LIN {X 0,Y 141.838,Z 280.43,A -85,B 0,C 180,E1 -24691.143,E2 -24691.143} C_VEL
LIN {X 0,Y 143.834,Z 282.618,A -85,B 0,C 180,E1 -24692.929,E2 -24692.929} C_VEL
LIN {X 0,Y 144.786,Z 284.534,A -85,B 0,C 180,E1 -24693.933,E2 -24693.933} C_VEL
LIN {X 0,Y 146.337,Z 286.504,A -85,B 0,C 180,E1 -24695.269,E2 -24695.269} C_VEL
LIN {X 0,Y 150.7,Z 294.3,A -85,B 0,C 180,E1 -24699.406,E2 -24699.406} C_VEL
LIN {X 0,Y 153.684,Z 300.784,A -85,B 0,C 180,E1 -24702.417,E2 -24702.417} C_VEL
LIN {X 0,Y 155.938,Z 307.443,A -85,B 0,C 180,E1 -24705.221,E2 -24705.221} C_VEL
LIN {X 0,Y 157.372,Z 314.543,A -85,B 0,C 180,E1 -24707.942,E2 -24707.942} C_VEL
LIN {X 0,Y 158.008,Z 322.698,A -85,B 0,C 180,E1 -24711.003,E2 -24711.003} C_VEL
LIN {X 0,Y 157.928,Z 328.022,A -85,B 0,C 180,E1 -24713.033,E2 -24713.033} C_VEL
LIN {X 0,Y 153.929,Z 337.234,A -85,B 0,C 180,E1 -24715.992,E2 -24715.992} C_VEL
LIN {X 0,Y 149.326,Z 346.098,A -85,B 0,C 180,E1 -24719.605,E2 -24719.605} C_VEL
LIN {X 0,Y 145.353,Z 353.222,A -85,B 0,C 180,E1 -24723.432,E2 -24723.432} C_VEL
LIN {X 0,Y 142.419,Z 358.024,A -85,B 0,C 180,E1 -24726.747,E2 -24726.747} C_VEL
LIN {X 0,Y 139.452,Z 362.688,A -85,B 0,C 180,E1 -24730.877,E2 -24730.877} C_VEL
LIN {X 0,Y 137.221,Z 366.245,A -85,B 0,C 180,E1 -24735.162,E2 -24735.162} C_VEL
LIN {X 0,Y 135.527,Z 369.09,A -85,B 0,C 180,E1 -24740.158,E2 -24740.158} C_VEL
LIN {X 0,Y 134.692,Z 370.431,A -85,B 0,C 180,E1 -24744.009,E2 -24744.009} C_VEL
LIN {X 0,Y 134.186,Z 371.258,A -85,B 0,C 180,E1 -24750,E2 -24750} C_VEL
LIN {X 0,Y 134.298,Z 371.063,A -85,B 0,C 180,E1 -24752.999,E2 -24752.999} C_VEL
LIN {X 0,Y 134.677,Z 370.479,A -85,B 0,C 180,E1 -24755.99,E2 -24755.99} C_VEL
LIN {X 0,Y 135.383,Z 369.328,A -85,B 0,C 180,E1 -24759.484,E2 -24759.484} C_VEL
LIN {X 0,Y 137.212,Z 366.372,A -85,B 0,C 180,E1 -24764.838,E2 -24764.838} C_VEL
LIN {X 0,Y 139.413,Z 362.863,A -85,B 0,C 180,E1 -24769.127,E2 -24769.127} C_VEL
LIN {X 0,Y 142.337,Z 358.248,A -85,B 0,C 180,E1 -24773.266,E2 -24773.266} C_VEL
LIN {X 0,Y 145.891,Z 352.391,A -85,B 0,C 180,E1 -24777.235,E2 -24777.235} C_VEL
LIN {X 0,Y 149.993,Z 345.085,A -85,B 0,C 180,E1 -24781.025,E2 -24781.025} C_VEL
LIN {X 0,Y 153.874,Z 337.64,A -85,B 0,C 180,E1 -24784.015,E2 -24784.015} C_VEL
LIN {X 0,Y 157.905,Z 328.606,A -85,B 0,C 180,E1 -24786.929,E2 -24786.929} C_VEL
LIN {X 0,Y 158.14,Z 324.518,A -85,B 0,C 180,E1 -24788.475,E2 -24788.475} C_VEL
LIN {X 0,Y 157.624,Z 316.205,A -85,B 0,C 180,E1 -24791.621,E2 -24791.621} C_VEL
LIN {X 0,Y 156.536,Z 309.758,A -85,B 0,C 180,E1 -24794.081,E2 -24794.081} C_VEL
LIN {X 0,Y 154.706,Z 303.491,A -85,B 0,C 180,E1 -24796.623,E2 -24796.623} C_VEL
LIN {X 0,Y 152.592,Z 298.134,A -85,B 0,C 180,E1 -24798.98,E2 -24798.98} C_VEL
LIN {X 0,Y 148.456,Z 290.276,A -85,B 0,C 180,E1 -24802.957,E2 -24802.957} C_VEL
LIN {X 0,Y 146.515,Z 286.687,A -85,B 0,C 180,E1 -24804.857,E2 -24804.857} C_VEL
LIN {X 0,Y 144.119,Z 283.245,A -85,B 0,C 180,E1 -24807.041,E2 -24807.041} C_VEL
LIN {X 0,Y 143.395,Z 281.959,A -85,B 0,C 180,E1 -24807.791,E2 -24807.791} C_VEL
LIN {X 0,Y 141.169,Z 279.417,A -85,B 0,C 180,E1 -24809.834,E2 -24809.834} C_VEL
LIN {X 0,Y 140.176,Z 277.103,A -85,B 0,C 180,E1 -24811.041,E2 -24811.041} C_VEL
LIN {X 0,Y 137.647,Z 275.103,A -85,B 0,C 180,E1 -24813.464,E2 -24813.464} C_VEL
LIN {X 0,Y 136.363,Z 272.838,A -85,B 0,C 180,E1 -24815.04,E2 -24815.04} C_VEL
LIN {X 0,Y 136.077,Z 271.532,A -85,B 0,C 180,E1 -24815.595,E2 -24815.595} C_VEL
LIN {X 0,Y 136.234,Z 271.511,A -85,B 0,C 180,E1 -24818.831,E2 -24818.831} C_VEL
LIN {X 0,Y 136.255,Z 271.507,A -85,B 0,C 180,E1 -24825.054,E2 -24825.054} C_VEL
LIN {X 0,Y 136.498,Z 271.479,A -85,B 0,C 180,E1 -24828.115,E2 -24828.115} C_VEL
LIN {X 0,Y 136.599,Z 271.47,A -85,B 0,C 180,E1 -24831.121,E2 -24831.121} C_VEL
LIN {X 0,Y 137.122,Z 271.399,A -85,B 0,C 180,E1 -24840,E2 -24840} C_VEL
LIN {X 0,Y 136.551,Z 271.512,A -85,B 0,C 180,E1 -24845.908,E2 -24845.908} C_VEL
LIN {X 0,Y 136.657,Z 272.118,A -85,B 0,C 180,E1 -24848.875,E2 -24848.875} C_VEL
LIN {X 0,Y 136.675,Z 272.963,A -85,B 0,C 180,E1 -24852.311,E2 -24852.311} C_VEL
LIN {X 0,Y 136.776,Z 274.589,A -85,B 0,C 180,E1 -24857.957,E2 -24857.957} C_VEL
LIN {X 0,Y 136.987,Z 276.148,A -85,B 0,C 180,E1 -24862.561,E2 -24862.561} C_VEL
LIN {X 0,Y 137.089,Z 277.31,A -85,B 0,C 180,E1 -24865.223,E2 -24865.223} C_VEL
LIN {X 0,Y 138.508,Z 280.757,A -85,B 0,C 180,E1 -24866.968,E2 -24866.968} C_VEL
LIN {X 0,Y 141.312,Z 284.181,A -85,B 0,C 180,E1 -24869.604,E2 -24869.604} C_VEL
LIN {X 0,Y 142.965,Z 287.925,A -85,B 0,C 180,E1 -24871.384,E2 -24871.384} C_VEL
LIN {X 0,Y 144.808,Z 290.602,A -85,B 0,C 180,E1 -24872.989,E2 -24872.989} C_VEL
LIN {X 0,Y 146.724,Z 294.699,A -85,B 0,C 180,E1 -24874.876,E2 -24874.876} C_VEL
LIN {X 0,Y 147.718,Z 296.419,A -85,B 0,C 180,E1 -24875.732,E2 -24875.732} C_VEL
LIN {X 0,Y 150.333,Z 302.421,A -85,B 0,C 180,E1 -24878.275,E2 -24878.275} C_VEL
LIN {X 0,Y 152.953,Z 308.925,A -85,B 0,C 180,E1 -24880.902,E2 -24880.902} C_VEL
LIN {X 0,Y 154.988,Z 316.134,A -85,B 0,C 180,E1 -24883.488,E2 -24883.488} C_VEL
LIN {X 0,Y 155.173,Z 324.491,A -85,B 0,C 180,E1 -24885.855,E2 -24885.855} C_VEL
LIN {X 0,Y 154.528,Z 334.205,A -85,B 0,C 180,E1 -24888.741,E2 -24888.741} C_VEL
LIN {X 0,Y 153.215,Z 343.18,A -85,B 0,C 180,E1 -24891.676,E2 -24891.676} C_VEL
LIN {X 0,Y 151.414,Z 350.973,A -85,B 0,C 180,E1 -24894.536,E2 -24894.536} C_VEL
LIN {X 0,Y 149.469,Z 355.913,A -85,B 0,C 180,E1 -24896.463,E2 -24896.463} C_VEL
LIN {X 0,Y 145.026,Z 364.22,A -85,B 0,C 180,E1 -24900.217,E2 -24900.217} C_VEL
LIN {X 0,Y 142.012,Z 369.919,A -85,B 0,C 180,E1 -24903.551,E2 -24903.551} C_VEL
LIN {X 0,Y 138.903,Z 375.489,A -85,B 0,C 180,E1 -24907.699,E2 -24907.699} C_VEL
LIN {X 0,Y 136.408,Z 379.863,A -85,B 0,C 180,E1 -24911.993,E2 -24911.993} C_VEL
LIN {X 0,Y 135.297,Z 382.196,A -85,B 0,C 180,E1 -24914.947,E2 -24914.947} C_VEL
LIN {X 0,Y 134.479,Z 384.089,A -85,B 0,C 180,E1 -24917.934,E2 -24917.934} C_VEL
LIN {X 0,Y 133.756,Z 386.544,A -85,B 0,C 180,E1 -24923.968,E2 -24923.968} C_VEL
LIN {X 0,Y 133.761,Z 387.177,A -85,B 0,C 180,E1 -24926.989,E2 -24926.989} C_VEL
LIN {X 0,Y 133.968,Z 387.409,A -85,B 0,C 180,E1 -24930,E2 -24930} C_VEL
LIN {X 0,Y 133.761,Z 387.108,A -85,B 0,C 180,E1 -24933.351,E2 -24933.351} C_VEL
LIN {X 0,Y 133.965,Z 385.487,A -85,B 0,C 180,E1 -24939.056,E2 -24939.056} C_VEL
LIN {X 0,Y 134.478,Z 384.046,A -85,B 0,C 180,E1 -24942.067,E2 -24942.067} C_VEL
LIN {X 0,Y 135.806,Z 381.043,A -85,B 0,C 180,E1 -24946.537,E2 -24946.537} C_VEL
LIN {X 0,Y 137.991,Z 377.008,A -85,B 0,C 180,E1 -24950.887,E2 -24950.887} C_VEL
LIN {X 0,Y 141.535,Z 370.828,A -85,B 0,C 180,E1 -24955.753,E2 -24955.753} C_VEL
LIN {X 0,Y 144.438,Z 365.325,A -85,B 0,C 180,E1 -24959.116,E2 -24959.116} C_VEL
LIN {X 0,Y 148.671,Z 357.234,A -85,B 0,C 180,E1 -24962.932,E2 -24962.932} C_VEL
LIN {X 0,Y 150.839,Z 352.476,A -85,B 0,C 180,E1 -24964.804,E2 -24964.804} C_VEL
LIN {X 0,Y 152.873,Z 344.49,A -85,B 0,C 180,E1 -24967.78,E2 -24967.78} C_VEL
LIN {X 0,Y 154.452,Z 333.906,A -85,B 0,C 180,E1 -24971.285,E2 -24971.285} C_VEL
LIN {X 0,Y 155.122,Z 324.256,A -85,B 0,C 180,E1 -24974.126,E2 -24974.126} C_VEL
LIN {X 0,Y 154.856,Z 315.67,A -85,B 0,C 180,E1 -24976.565,E2 -24976.565} C_VEL
LIN {X 0,Y 152.839,Z 308.741,A -85,B 0,C 180,E1 -24979.061,E2 -24979.061} C_VEL
LIN {X 0,Y 149.573,Z 300.435,A -85,B 0,C 180,E1 -24982.35,E2 -24982.35} C_VEL
LIN {X 0,Y 146.945,Z 294.996,A -85,B 0,C 180,E1 -24984.787,E2 -24984.787} C_VEL
LIN {X 0,Y 144.827,Z 290.683,A -85,B 0,C 180,E1 -24986.808,E2 -24986.808} C_VEL
LIN {X 0,Y 144.013,Z 289.318,A -85,B 0,C 180,E1 -24987.533,E2 -24987.533} C_VEL
LIN {X 0,Y 141.84,Z 285.601,A -85,B 0,C 180,E1 -24989.581,E2 -24989.581} C_VEL
LIN {X 0,Y 141.162,Z 283.864,A -85,B 0,C 180,E1 -24990.344,E2 -24990.344} C_VEL
LIN {X 0,Y 139.957,Z 282.669,A -85,B 0,C 180,E1 -24991.39,E2 -24991.39} C_VEL
LIN {X 0,Y 137.115,Z 279.685,A -85,B 0,C 180,E1 -24994.165,E2 -24994.165} C_VEL
LIN {X 0,Y 134.138,Z 277.82,A -85,B 0,C 180,E1 -24997.154,E2 -24997.154} C_VEL
LIN {X 0,Y 130.283,Z 276.151,A -85,B 0,C 180,E1 -25001.971,E2 -25001.971} C_VEL
LIN {X 0,Y 129.764,Z 275.679,A -85,B 0,C 180,E1 -25003.674,E2 -25003.674} C_VEL
LIN {X 0,Y 129.767,Z 274.653,A -85,B 0,C 180,E1 -25007.489,E2 -25007.489} C_VEL
LIN {X 0,Y 129.743,Z 273.911,A -85,B 0,C 180,E1 -25010.648,E2 -25010.648} C_VEL
LIN {X 0,Y 129.745,Z 272.681,A -85,B 0,C 180,E1 -25016.895,E2 -25016.895} C_VEL
LIN {X 0,Y 130.078,Z 272.28,A -85,B 0,C 180,E1 -25020,E2 -25020} C_VEL
LIN {X 0,Y 129.474,Z 272.354,A -85,B 0,C 180,E1 -25029.372,E2 -25029.372} C_VEL
LIN {X 0,Y 129.302,Z 272.376,A -85,B 0,C 180,E1 -25032.557,E2 -25032.557} C_VEL
LIN {X 0,Y 129.139,Z 272.538,A -85,B 0,C 180,E1 -25036.907,E2 -25036.907} C_VEL
LIN {X 0,Y 130.094,Z 275.183,A -85,B 0,C 180,E1 -25039.016,E2 -25039.016} C_VEL
LIN {X 0,Y 132.779,Z 277.797,A -85,B 0,C 180,E1 -25042.857,E2 -25042.857} C_VEL
LIN {X 0,Y 133.593,Z 278.36,A -85,B 0,C 180,E1 -25043.855,E2 -25043.855} C_VEL
LIN {X 0,Y 135.086,Z 281.391,A -85,B 0,C 180,E1 -25046.039,E2 -25046.039} C_VEL
LIN {X 0,Y 137.339,Z 283.753,A -85,B 0,C 180,E1 -25048.564,E2 -25048.564} C_VEL
LIN {X 0,Y 138.822,Z 286.608,A -85,B 0,C 180,E1 -25050.415,E2 -25050.415} C_VEL
LIN {X 0,Y 140.029,Z 287.941,A -85,B 0,C 180,E1 -25051.634,E2 -25051.634} C_VEL
LIN {X 0,Y 143.078,Z 293.333,A -85,B 0,C 180,E1 -25055.044,E2 -25055.044} C_VEL
LIN {X 0,Y 146.358,Z 299.552,A -85,B 0,C 180,E1 -25058.627,E2 -25058.627} C_VEL
LIN {X 0,Y 149.095,Z 306.237,A -85,B 0,C 180,E1 -25061.958,E2 -25061.958} C_VEL
LIN {X 0,Y 150.661,Z 311.65,A -85,B 0,C 180,E1 -25064.405,E2 -25064.405} C_VEL
LIN {X 0,Y 151.716,Z 318.596,A -85,B 0,C 180,E1 -25067.284,E2 -25067.284} C_VEL
LIN {X 0,Y 151.973,Z 326.544,A -85,B 0,C 180,E1 -25070.516,E2 -25070.516} C_VEL
LIN {X 0,Y 151.59,Z 330.298,A -85,B 0,C 180,E1 -25072.014,E2 -25072.014} C_VEL
LIN {X 0,Y 147.276,Z 339.276,A -85,B 0,C 180,E1 -25075.065,E2 -25075.065} C_VEL
LIN {X 0,Y 142.529,Z 347.845,A -85,B 0,C 180,E1 -25078.818,E2 -25078.818} C_VEL
LIN {X 0,Y 138.376,Z 354.671,A -85,B 0,C 180,E1 -25082.799,E2 -25082.799} C_VEL
LIN {X 0,Y 134.808,Z 360.132,A -85,B 0,C 180,E1 -25086.983,E2 -25086.983} C_VEL
LIN {X 0,Y 131.9,Z 364.413,A -85,B 0,C 180,E1 -25091.355,E2 -25091.355} C_VEL
LIN {X 0,Y 130.388,Z 366.673,A -85,B 0,C 180,E1 -25094.365,E2 -25094.365} C_VEL
LIN {X 0,Y 128.443,Z 369.696,A -85,B 0,C 180,E1 -25100.033,E2 -25100.033} C_VEL
LIN {X 0,Y 127.658,Z 370.857,A -85,B 0,C 180,E1 -25103.678,E2 -25103.678} C_VEL
LIN {X 0,Y 127.109,Z 371.684,A -85,B 0,C 180,E1 -25110,E2 -25110} C_VEL
LIN {X 0,Y 127.232,Z 371.489,A -85,B 0,C 180,E1 -25113.166,E2 -25113.166} C_VEL
LIN {X 0,Y 127.642,Z 370.904,A -85,B 0,C 180,E1 -25116.322,E2 -25116.322} C_VEL
LIN {X 0,Y 128.308,Z 369.89,A -85,B 0,C 180,E1 -25119.618,E2 -25119.618} C_VEL
LIN {X 0,Y 129.162,Z 368.6,A -85,B 0,C 180,E1 -25122.571,E2 -25122.571} C_VEL
LIN {X 0,Y 131.084,Z 365.752,A -85,B 0,C 180,E1 -25127.15,E2 -25127.15} C_VEL
LIN {X 0,Y 133.683,Z 361.885,A -85,B 0,C 180,E1 -25131.592,E2 -25131.592} C_VEL
LIN {X 0,Y 137.004,Z 356.887,A -85,B 0,C 180,E1 -25135.851,E2 -25135.851} C_VEL
LIN {X 0,Y 140.922,Z 350.586,A -85,B 0,C 180,E1 -25139.915,E2 -25139.915} C_VEL
LIN {X 0,Y 145.569,Z 342.69,A -85,B 0,C 180,E1 -25143.725,E2 -25143.725} C_VEL
LIN {X 0,Y 149.694,Z 334.74,A -85,B 0,C 180,E1 -25146.724,E2 -25146.724} C_VEL
LIN {X 0,Y 151.705,Z 330.332,A -85,B 0,C 180,E1 -25148.141,E2 -25148.141} C_VEL
LIN {X 0,Y 152.052,Z 328.068,A -85,B 0,C 180,E1 -25149.031,E2 -25149.031} C_VEL
LIN {X 0,Y 151.927,Z 320.219,A -85,B 0,C 180,E1 -25152.256,E2 -25152.256} C_VEL
LIN {X 0,Y 151.152,Z 313.899,A -85,B 0,C 180,E1 -25154.841,E2 -25154.841} C_VEL
LIN {X 0,Y 149.884,Z 308.565,A -85,B 0,C 180,E1 -25157.164,E2 -25157.164} C_VEL
LIN {X 0,Y 147.852,Z 302.837,A -85,B 0,C 180,E1 -25159.902,E2 -25159.902} C_VEL
LIN {X 0,Y 144.052,Z 295.111,A -85,B 0,C 180,E1 -25164.165,E2 -25164.165} C_VEL
LIN {X 0,Y 140.337,Z 288.305,A -85,B 0,C 180,E1 -25168.359,E2 -25168.359} C_VEL
LIN {X 0,Y 137.933,Z 285.126,A -85,B 0,C 180,E1 -25170.945,E2 -25170.945} C_VEL
LIN {X 0,Y 137.08,Z 283.29,A -85,B 0,C 180,E1 -25172.106,E2 -25172.106} C_VEL
LIN {X 0,Y 134.839,Z 281.062,A -85,B 0,C 180,E1 -25174.635,E2 -25174.635} C_VEL
LIN {X 0,Y 133.47,Z 278.105,A -85,B 0,C 180,E1 -25176.739,E2 -25176.739} C_VEL
LIN {X 0,Y 130.52,Z 275.806,A -85,B 0,C 180,E1 -25180.743,E2 -25180.743} C_VEL
LIN {X 0,Y 129.286,Z 273.228,A -85,B 0,C 180,E1 -25183.214,E2 -25183.214} C_VEL
LIN {X 0,Y 129.151,Z 272.397,A -85,B 0,C 180,E1 -25183.806,E2 -25183.806} C_VEL
LIN {X 0,Y 129.417,Z 272.362,A -85,B 0,C 180,E1 -25187.819,E2 -25187.819} C_VEL
LIN {X 0,Y 129.523,Z 272.351,A -85,B 0,C 180,E1 -25190.631,E2 -25190.631} C_VEL
LIN {X 0,Y 130.078,Z 272.277,A -85,B 0,C 180,E1 -25200,E2 -25200} C_VEL
LIN {X 0,Y 129.675,Z 273.326,A -85,B 0,C 180,E1 -25206.223,E2 -25206.223} C_VEL
LIN {X 0,Y 129.753,Z 273.959,A -85,B 0,C 180,E1 -25209.352,E2 -25209.352} C_VEL
LIN {X 0,Y 129.747,Z 274.803,A -85,B 0,C 180,E1 -25212.837,E2 -25212.837} C_VEL
LIN {X 0,Y 129.845,Z 276.105,A -85,B 0,C 180,E1 -25217.218,E2 -25217.218} C_VEL
LIN {X 0,Y 131.083,Z 279.36,A -85,B 0,C 180,E1 -25219.578,E2 -25219.578} C_VEL
LIN {X 0,Y 134.498,Z 283.59,A -85,B 0,C 180,E1 -25224.067,E2 -25224.067} C_VEL
LIN {X 0,Y 136.042,Z 287.254,A -85,B 0,C 180,E1 -25226.253,E2 -25226.253} C_VEL
LIN {X 0,Y 138.127,Z 290.066,A -85,B 0,C 180,E1 -25228.49,E2 -25228.49} C_VEL
LIN {X 0,Y 139.661,Z 293.716,A -85,B 0,C 180,E1 -25230.422,E2 -25230.422} C_VEL
LIN {X 0,Y 140.848,Z 295.505,A -85,B 0,C 180,E1 -25231.598,E2 -25231.598} C_VEL
LIN {X 0,Y 142.604,Z 299.67,A -85,B 0,C 180,E1 -25233.672,E2 -25233.672} C_VEL
LIN {X 0,Y 143.862,Z 302.367,A -85,B 0,C 180,E1 -25235.031,E2 -25235.031} C_VEL
LIN {X 0,Y 146.829,Z 309.908,A -85,B 0,C 180,E1 -25238.481,E2 -25238.481} C_VEL
LIN {X 0,Y 148.984,Z 316.8,A -85,B 0,C 180,E1 -25241.332,E2 -25241.332} C_VEL
LIN {X 0,Y 149.548,Z 319.996,A -85,B 0,C 180,E1 -25242.497,E2 -25242.497} C_VEL
LIN {X 0,Y 149.194,Z 329.568,A -85,B 0,C 180,E1 -25245.436,E2 -25245.436} C_VEL
LIN {X 0,Y 148.095,Z 338.521,A -85,B 0,C 180,E1 -25248.365,E2 -25248.365} C_VEL
LIN {X 0,Y 146.414,Z 346.871,A -85,B 0,C 180,E1 -25251.391,E2 -25251.391} C_VEL
LIN {X 0,Y 144.318,Z 353.893,A -85,B 0,C 180,E1 -25254.241,E2 -25254.241} C_VEL
LIN {X 0,Y 139.599,Z 362.547,A -85,B 0,C 180,E1 -25258.088,E2 -25258.088} C_VEL
LIN {X 0,Y 135.603,Z 369.487,A -85,B 0,C 180,E1 -25262.196,E2 -25262.196} C_VEL
LIN {X 0,Y 132.316,Z 375.06,A -85,B 0,C 180,E1 -25266.524,E2 -25266.524} C_VEL
LIN {X 0,Y 129.641,Z 379.435,A -85,B 0,C 180,E1 -25271.019,E2 -25271.019} C_VEL
LIN {X 0,Y 128.409,Z 381.766,A -85,B 0,C 180,E1 -25274.118,E2 -25274.118} C_VEL
LIN {X 0,Y 127.496,Z 383.659,A -85,B 0,C 180,E1 -25277.262,E2 -25277.262} C_VEL
LIN {X 0,Y 126.695,Z 386.117,A -85,B 0,C 180,E1 -25283.631,E2 -25283.631} C_VEL
LIN {X 0,Y 126.699,Z 386.751,A -85,B 0,C 180,E1 -25286.821,E2 -25286.821} C_VEL
LIN {X 0,Y 126.888,Z 386.983,A -85,B 0,C 180,E1 -25290,E2 -25290} C_VEL
LIN {X 0,Y 126.699,Z 386.738,A -85,B 0,C 180,E1 -25293.18,E2 -25293.18} C_VEL
LIN {X 0,Y 126.695,Z 386.095,A -85,B 0,C 180,E1 -25296.37,E2 -25296.37} C_VEL
LIN {X 0,Y 126.929,Z 385.057,A -85,B 0,C 180,E1 -25299.562,E2 -25299.562} C_VEL
LIN {X 0,Y 127.496,Z 383.615,A -85,B 0,C 180,E1 -25302.739,E2 -25302.739} C_VEL
LIN {X 0,Y 128.96,Z 380.611,A -85,B 0,C 180,E1 -25307.442,E2 -25307.442} C_VEL
LIN {X 0,Y 131.354,Z 376.577,A -85,B 0,C 180,E1 -25311.996,E2 -25311.996} C_VEL
LIN {X 0,Y 135.105,Z 370.394,A -85,B 0,C 180,E1 -25317.076,E2 -25317.076} C_VEL
LIN {X 0,Y 138.893,Z 363.644,A -85,B 0,C 180,E1 -25321.242,E2 -25321.242} C_VEL
LIN {X 0,Y 143.558,Z 355.303,A -85,B 0,C 180,E1 -25325.117,E2 -25325.117} C_VEL
LIN {X 0,Y 145.884,Z 348.483,A -85,B 0,C 180,E1 -25327.897,E2 -25327.897} C_VEL
LIN {X 0,Y 147.792,Z 339.678,A -85,B 0,C 180,E1 -25331.15,E2 -25331.15} C_VEL
LIN {X 0,Y 149.157,Z 329.357,A -85,B 0,C 180,E1 -25334.536,E2 -25334.536} C_VEL
LIN {X 0,Y 149.45,Z 319.741,A -85,B 0,C 180,E1 -25337.495,E2 -25337.495} C_VEL
LIN {X 0,Y 148.435,Z 315.085,A -85,B 0,C 180,E1 -25339.25,E2 -25339.25} C_VEL
LIN {X 0,Y 145.355,Z 305.938,A -85,B 0,C 180,E1 -25343.125,E2 -25343.125} C_VEL
LIN {X 0,Y 143.152,Z 300.592,A -85,B 0,C 180,E1 -25345.626,E2 -25345.626} C_VEL
LIN {X 0,Y 140.261,Z 294.62,A -85,B 0,C 180,E1 -25348.781,E2 -25348.781} C_VEL
LIN {X 0,Y 138.297,Z 290.655,A -85,B 0,C 180,E1 -25351.03,E2 -25351.03} C_VEL
LIN {X 0,Y 137.714,Z 289.47,A -85,B 0,C 180,E1 -25351.728,E2 -25351.728} C_VEL
LIN {X 0,Y 135.243,Z 285.741,A -85,B 0,C 180,E1 -25354.511,E2 -25354.511} C_VEL
LIN {X 0,Y 134.299,Z 283.255,A -85,B 0,C 180,E1 -25355.915,E2 -25355.915} C_VEL
LIN {X 0,Y 131,Z 279.223,A -85,B 0,C 180,E1 -25360.205,E2 -25360.205} C_VEL
LIN {X 0,Y 129.885,Z 276.326,A -85,B 0,C 180,E1 -25362.28,E2 -25362.28} C_VEL
LIN {X 0,Y 129.813,Z 275.958,A -85,B 0,C 180,E1 -25362.677,E2 -25362.677} C_VEL
LIN {X 0,Y 129.764,Z 275.679,A -85,B 0,C 180,E1 -25363.674,E2 -25363.674} C_VEL
LIN {X 0,Y 129.141,Z 275.368,A -85,B 0,C 180,E1 -25366.26,E2 -25366.26} C_VEL
LIN {X 0,Y 127.775,Z 275.626,A -85,B 0,C 180,E1 -25368.835,E2 -25368.835} C_VEL
LIN {X 0,Y 124.576,Z 276.386,A -85,B 0,C 180,E1 -25374.087,E2 -25374.087} C_VEL
LIN {X 0,Y 123.628,Z 276.153,A -85,B 0,C 180,E1 -25376.82,E2 -25376.82} C_VEL
LIN {X 0,Y 123.523,Z 275.89,A -85,B 0,C 180,E1 -25377.737,E2 -25377.737} C_VEL
LIN {X 0,Y 123.527,Z 275.06,A -85,B 0,C 180,E1 -25380,E2 -25380} C_VEL
LIN {X 0,Y 127.17,Z 279.374,A -85,B 0,C 180,E1 -25396.041,E2 -25396.041} C_VEL
LIN {X 0,Y 128.279,Z 282.184,A -85,B 0,C 180,E1 -25398.776,E2 -25398.776} C_VEL
LIN {X 0,Y 131.018,Z 284.995,A -85,B 0,C 180,E1 -25403.095,E2 -25403.095} C_VEL
LIN {X 0,Y 132.245,Z 287.538,A -85,B 0,C 180,E1 -25405.16,E2 -25405.16} C_VEL
LIN {X 0,Y 134.392,Z 290.483,A -85,B 0,C 180,E1 -25408.077,E2 -25408.077} C_VEL
LIN {X 0,Y 137.055,Z 294.959,A -85,B 0,C 180,E1 -25411.583,E2 -25411.583} C_VEL
LIN {X 0,Y 140.497,Z 301.611,A -85,B 0,C 180,E1 -25415.999,E2 -25415.999} C_VEL
LIN {X 0,Y 143.176,Z 307.908,A -85,B 0,C 180,E1 -25419.653,E2 -25419.653} C_VEL
LIN {X 0,Y 144.959,Z 313.997,A -85,B 0,C 180,E1 -25422.747,E2 -25422.747} C_VEL
LIN {X 0,Y 145.971,Z 321.706,A -85,B 0,C 180,E1 -25426.237,E2 -25426.237} C_VEL
LIN {X 0,Y 145.952,Z 329.06,A -85,B 0,C 180,E1 -25429.455,E2 -25429.455} C_VEL
LIN {X 0,Y 145.692,Z 331.463,A -85,B 0,C 180,E1 -25430.518,E2 -25430.518} C_VEL
LIN {X 0,Y 141.535,Z 339.705,A -85,B 0,C 180,E1 -25433.425,E2 -25433.425} C_VEL
LIN {X 0,Y 136.519,Z 348.274,A -85,B 0,C 180,E1 -25437.279,E2 -25437.279} C_VEL
LIN {X 0,Y 132.108,Z 355.1,A -85,B 0,C 180,E1 -25441.393,E2 -25441.393} C_VEL
LIN {X 0,Y 128.306,Z 360.561,A -85,B 0,C 180,E1 -25445.743,E2 -25445.743} C_VEL
LIN {X 0,Y 125.194,Z 364.842,A -85,B 0,C 180,E1 -25450.316,E2 -25450.316} C_VEL
LIN {X 0,Y 123.574,Z 367.101,A -85,B 0,C 180,E1 -25453.479,E2 -25453.479} C_VEL
LIN {X 0,Y 122.308,Z 368.932,A -85,B 0,C 180,E1 -25456.711,E2 -25456.711} C_VEL
LIN {X 0,Y 121.362,Z 370.304,A -85,B 0,C 180,E1 -25459.995,E2 -25459.995} C_VEL
LIN {X 0,Y 120.172,Z 371.887,A -85,B 0,C 180,E1 -25466.647,E2 -25466.647} C_VEL
LIN {X 0,Y 120.034,Z 372.11,A -85,B 0,C 180,E1 -25470,E2 -25470} C_VEL
LIN {X 0,Y 120.169,Z 371.914,A -85,B 0,C 180,E1 -25473.352,E2 -25473.352} C_VEL
LIN {X 0,Y 121.272,Z 370.416,A -85,B 0,C 180,E1 -25479.871,E2 -25479.871} C_VEL
LIN {X 0,Y 122.259,Z 369.026,A -85,B 0,C 180,E1 -25483.293,E2 -25483.293} C_VEL
LIN {X 0,Y 124.337,Z 366.177,A -85,B 0,C 180,E1 -25488.112,E2 -25488.112} C_VEL
LIN {X 0,Y 127.129,Z 362.31,A -85,B 0,C 180,E1 -25492.766,E2 -25492.766} C_VEL
LIN {X 0,Y 130.664,Z 357.312,A -85,B 0,C 180,E1 -25497.206,E2 -25497.206} C_VEL
LIN {X 0,Y 134.836,Z 351.01,A -85,B 0,C 180,E1 -25501.414,E2 -25501.414} C_VEL
LIN {X 0,Y 139.744,Z 343.113,A -85,B 0,C 180,E1 -25505.335,E2 -25505.335} C_VEL
LIN {X 0,Y 144.368,Z 334.556,A -85,B 0,C 180,E1 -25508.624,E2 -25508.624} C_VEL
LIN {X 0,Y 145.801,Z 331.579,A -85,B 0,C 180,E1 -25509.603,E2 -25509.603} C_VEL
LIN {X 0,Y 146.129,Z 323.848,A -85,B 0,C 180,E1 -25513.021,E2 -25513.021} C_VEL
LIN {X 0,Y 145.701,Z 317.971,A -85,B 0,C 180,E1 -25515.621,E2 -25515.621} C_VEL
LIN {X 0,Y 144.719,Z 312.913,A -85,B 0,C 180,E1 -25518.014,E2 -25518.014} C_VEL
LIN {X 0,Y 142.827,Z 306.924,A -85,B 0,C 180,E1 -25521.143,E2 -25521.143} C_VEL
LIN {X 0,Y 139.531,Z 299.744,A -85,B 0,C 180,E1 -25525.483,E2 -25525.483} C_VEL
LIN {X 0,Y 136.844,Z 294.313,A -85,B 0,C 180,E1 -25529.097,E2 -25529.097} C_VEL
LIN {X 0,Y 133.533,Z 289.129,A -85,B 0,C 180,E1 -25533.473,E2 -25533.473} C_VEL
LIN {X 0,Y 131.521,Z 286.241,A -85,B 0,C 180,E1 -25536.373,E2 -25536.373} C_VEL
LIN {X 0,Y 130.946,Z 284.669,A -85,B 0,C 180,E1 -25537.517,E2 -25537.517} C_VEL
LIN {X 0,Y 128.233,Z 282.087,A -85,B 0,C 180,E1 -25541.837,E2 -25541.837} C_VEL
LIN {X 0,Y 127.098,Z 279.172,A -85,B 0,C 180,E1 -25544.772,E2 -25544.772} C_VEL
LIN {X 0,Y 123.746,Z 275.561,A -85,B 0,C 180,E1 -25560,E2 -25560} C_VEL
LIN {X 0,Y 125.158,Z 279.582,A -85,B 0,C 180,E1 -25570.106,E2 -25570.106} C_VEL
LIN {X 0,Y 127.849,Z 282.799,A -85,B 0,C 180,E1 -25576.261,E2 -25576.261} C_VEL
LIN {X 0,Y 129.097,Z 286.174,A -85,B 0,C 180,E1 -25579.065,E2 -25579.065} C_VEL
LIN {X 0,Y 131.728,Z 289.94,A -85,B 0,C 180,E1 -25583.067,E2 -25583.067} C_VEL
LIN {X 0,Y 133.489,Z 294.019,A -85,B 0,C 180,E1 -25585.85,E2 -25585.85} C_VEL
LIN {X 0,Y 135.033,Z 296.889,A -85,B 0,C 180,E1 -25587.932,E2 -25587.932} C_VEL
LIN {X 0,Y 137.653,Z 302.869,A -85,B 0,C 180,E1 -25591.506,E2 -25591.506} C_VEL
LIN {X 0,Y 139.843,Z 308.261,A -85,B 0,C 180,E1 -25594.429,E2 -25594.429} C_VEL
LIN {X 0,Y 142.769,Z 316.989,A -85,B 0,C 180,E1 -25598.647,E2 -25598.647} C_VEL
LIN {X 0,Y 144.037,Z 323.047,A -85,B 0,C 180,E1 -25601.212,E2 -25601.212} C_VEL
LIN {X 0,Y 143.311,Z 332.184,A -85,B 0,C 180,E1 -25604.249,E2 -25604.249} C_VEL
LIN {X 0,Y 141.669,Z 341.847,A -85,B 0,C 180,E1 -25607.689,E2 -25607.689} C_VEL
LIN {X 0,Y 139.539,Z 350.081,A -85,B 0,C 180,E1 -25610.981,E2 -25610.981} C_VEL
LIN {X 0,Y 137.751,Z 355.055,A -85,B 0,C 180,E1 -25613.168,E2 -25613.168} C_VEL
LIN {X 0,Y 132.813,Z 363.363,A -85,B 0,C 180,E1 -25617.154,E2 -25617.154} C_VEL
LIN {X 0,Y 128.715,Z 370.082,A -85,B 0,C 180,E1 -25621.461,E2 -25621.461} C_VEL
LIN {X 0,Y 124.779,Z 376.237,A -85,B 0,C 180,E1 -25626.78,E2 -25626.78} C_VEL
LIN {X 0,Y 122.163,Z 380.245,A -85,B 0,C 180,E1 -25631.554,E2 -25631.554} C_VEL
LIN {X 0,Y 120.545,Z 383.23,A -85,B 0,C 180,E1 -25636.514,E2 -25636.514} C_VEL
LIN {X 0,Y 119.634,Z 385.689,A -85,B 0,C 180,E1 -25643.253,E2 -25643.253} C_VEL
LIN {X 0,Y 119.614,Z 386.409,A -85,B 0,C 180,E1 -25647.251,E2 -25647.251} C_VEL
LIN {X 0,Y 119.791,Z 386.555,A -85,B 0,C 180,E1 -25650,E2 -25650} C_VEL
LIN {X 0,Y 119.602,Z 386.31,A -85,B 0,C 180,E1 -25653.369,E2 -25653.369} C_VEL
LIN {X 0,Y 119.633,Z 385.666,A -85,B 0,C 180,E1 -25656.748,E2 -25656.748} C_VEL
LIN {X 0,Y 119.918,Z 384.628,A -85,B 0,C 180,E1 -25660.127,E2 -25660.127} C_VEL
LIN {X 0,Y 120.544,Z 383.185,A -85,B 0,C 180,E1 -25663.487,E2 -25663.487} C_VEL
LIN {X 0,Y 122.163,Z 380.18,A -85,B 0,C 180,E1 -25668.447,E2 -25668.447} C_VEL
LIN {X 0,Y 124.772,Z 376.147,A -85,B 0,C 180,E1 -25673.222,E2 -25673.222} C_VEL
LIN {X 0,Y 128.748,Z 369.96,A -85,B 0,C 180,E1 -25678.532,E2 -25678.532} C_VEL
LIN {X 0,Y 132.823,Z 363.211,A -85,B 0,C 180,E1 -25682.845,E2 -25682.845} C_VEL
LIN {X 0,Y 137.722,Z 354.866,A -85,B 0,C 180,E1 -25686.843,E2 -25686.843} C_VEL
LIN {X 0,Y 140.069,Z 348.03,A -85,B 0,C 180,E1 -25689.773,E2 -25689.773} C_VEL
LIN {X 0,Y 142.02,Z 339.546,A -85,B 0,C 180,E1 -25693.07,E2 -25693.07} C_VEL
LIN {X 0,Y 143.452,Z 330.399,A -85,B 0,C 180,E1 -25696.242,E2 -25696.242} C_VEL
LIN {X 0,Y 143.929,Z 322.484,A -85,B 0,C 180,E1 -25698.888,E2 -25698.888} C_VEL
LIN {X 0,Y 142.79,Z 317.205,A -85,B 0,C 180,E1 -25701.132,E2 -25701.132} C_VEL
LIN {X 0,Y 140.251,Z 309.446,A -85,B 0,C 180,E1 -25704.812,E2 -25704.812} C_VEL
LIN {X 0,Y 137.11,Z 301.16,A -85,B 0,C 180,E1 -25709.164,E2 -25709.164} C_VEL
LIN {X 0,Y 134.907,Z 296.535,A -85,B 0,C 180,E1 -25712.04,E2 -25712.04} C_VEL
LIN {X 0,Y 134.619,Z 295.517,A -85,B 0,C 180,E1 -25712.564,E2 -25712.564} C_VEL
LIN {X 0,Y 132.24,Z 291.58,A -85,B 0,C 180,E1 -25715.677,E2 -25715.677} C_VEL
LIN {X 0,Y 131.526,Z 289.422,A -85,B 0,C 180,E1 -25717,E2 -25717} C_VEL
LIN {X 0,Y 128.551,Z 285.144,A -85,B 0,C 180,E1 -25721.575,E2 -25721.575} C_VEL
LIN {X 0,Y 127.703,Z 282.512,A -85,B 0,C 180,E1 -25723.618,E2 -25723.618} C_VEL
LIN {X 0,Y 123.651,Z 276.594,A -85,B 0,C 180,E1 -25735.926,E2 -25735.926} C_VEL
LIN {X 0,Y 123.523,Z 275.89,A -85,B 0,C 180,E1 -25737.737,E2 -25737.737} C_VEL
LIN {X 0,Y 123.413,Z 275.78,A -85,B 0,C 180,E1 -25739.54,E2 -25739.54} C_VEL
LIN {X 0,Y 123.273,Z 276.486,A -85,B 0,C 180,E1 -25741.325,E2 -25741.325} C_VEL
LIN {X 0,Y 123.004,Z 279.35,A -85,B 0,C 180,E1 -25744.775,E2 -25744.775} C_VEL
LIN {X 0,Y 123.01,Z 283.56,A -85,B 0,C 180,E1 -25749.12,E2 -25749.12} C_VEL
LIN {X 0,Y 123.594,Z 285.061,A -85,B 0,C 180,E1 -25751.844,E2 -25751.844} C_VEL
LIN {X 0,Y 124.951,Z 286.092,A -85,B 0,C 180,E1 -25755.287,E2 -25755.287} C_VEL
LIN {X 0,Y 125.809,Z 288.538,A -85,B 0,C 180,E1 -25757.895,E2 -25757.895} C_VEL
LIN {X 0,Y 128.264,Z 291.709,A -85,B 0,C 180,E1 -25762.554,E2 -25762.554} C_VEL
LIN {X 0,Y 130.936,Z 296.317,A -85,B 0,C 180,E1 -25767.145,E2 -25767.145} C_VEL
LIN {X 0,Y 133.336,Z 300.853,A -85,B 0,C 180,E1 -25770.925,E2 -25770.925} C_VEL
LIN {X 0,Y 136.283,Z 307.243,A -85,B 0,C 180,E1 -25775.462,E2 -25775.462} C_VEL
LIN {X 0,Y 138.523,Z 313.588,A -85,B 0,C 180,E1 -25779.362,E2 -25779.362} C_VEL
LIN {X 0,Y 139.864,Z 319.836,A -85,B 0,C 180,E1 -25782.716,E2 -25782.716} C_VEL
LIN {X 0,Y 140.205,Z 326.64,A -85,B 0,C 180,E1 -25786.011,E2 -25786.011} C_VEL
LIN {X 0,Y 139.638,Z 333.288,A -85,B 0,C 180,E1 -25789.133,E2 -25789.133} C_VEL
LIN {X 0,Y 135.016,Z 341.717,A -85,B 0,C 180,E1 -25792.292,E2 -25792.292} C_VEL
LIN {X 0,Y 129.8,Z 349.922,A -85,B 0,C 180,E1 -25796.29,E2 -25796.29} C_VEL
LIN {X 0,Y 125.929,Z 355.529,A -85,B 0,C 180,E1 -25799.848,E2 -25799.848} C_VEL
LIN {X 0,Y 121.872,Z 360.99,A -85,B 0,C 180,E1 -25804.373,E2 -25804.373} C_VEL
LIN {X 0,Y 118.546,Z 365.27,A -85,B 0,C 180,E1 -25809.162,E2 -25809.162} C_VEL
LIN {X 0,Y 116.785,Z 367.529,A -85,B 0,C 180,E1 -25812.488,E2 -25812.488} C_VEL
LIN {X 0,Y 115.426,Z 369.359,A -85,B 0,C 180,E1 -25815.903,E2 -25815.903} C_VEL
LIN {X 0,Y 114.337,Z 370.793,A -85,B 0,C 180,E1 -25819.572,E2 -25819.572} C_VEL
LIN {X 0,Y 113.112,Z 372.313,A -85,B 0,C 180,E1 -25826.437,E2 -25826.437} C_VEL
LIN {X 0,Y 112.96,Z 372.536,A -85,B 0,C 180,E1 -25829.999,E2 -25829.999} C_VEL
LIN {X 0,Y 113.109,Z 372.34,A -85,B 0,C 180,E1 -25833.562,E2 -25833.562} C_VEL
LIN {X 0,Y 114.136,Z 371.037,A -85,B 0,C 180,E1 -25839.864,E2 -25839.864} C_VEL
LIN {X 0,Y 115.364,Z 369.453,A -85,B 0,C 180,E1 -25844.103,E2 -25844.103} C_VEL
LIN {X 0,Y 117.608,Z 366.604,A -85,B 0,C 180,E1 -25849.188,E2 -25849.188} C_VEL
LIN {X 0,Y 120.636,Z 362.735,A -85,B 0,C 180,E1 -25854.067,E2 -25854.067} C_VEL
LIN {X 0,Y 124.407,Z 357.737,A -85,B 0,C 180,E1 -25858.697,E2 -25858.697} C_VEL
LIN {X 0,Y 128.853,Z 351.434,A -85,B 0,C 180,E1 -25863.054,E2 -25863.054} C_VEL
LIN {X 0,Y 134.034,Z 343.537,A -85,B 0,C 180,E1 -25867.084,E2 -25867.084} C_VEL
LIN {X 0,Y 138.71,Z 335.346,A -85,B 0,C 180,E1 -25870.319,E2 -25870.319} C_VEL
LIN {X 0,Y 139.761,Z 333.307,A -85,B 0,C 180,E1 -25871.036,E2 -25871.036} C_VEL
LIN {X 0,Y 140.276,Z 326.898,A -85,B 0,C 180,E1 -25874.069,E2 -25874.069} C_VEL
LIN {X 0,Y 140.129,Z 321.452,A -85,B 0,C 180,E1 -25876.694,E2 -25876.694} C_VEL
LIN {X 0,Y 139.031,Z 315.411,A -85,B 0,C 180,E1 -25879.867,E2 -25879.867} C_VEL
LIN {X 0,Y 137.351,Z 309.995,A -85,B 0,C 180,E1 -25883.042,E2 -25883.042} C_VEL
LIN {X 0,Y 134.575,Z 303.28,A -85,B 0,C 180,E1 -25887.547,E2 -25887.547} C_VEL
LIN {X 0,Y 133.095,Z 300.091,A -85,B 0,C 180,E1 -25889.891,E2 -25889.891} C_VEL
LIN {X 0,Y 130.206,Z 295.084,A -85,B 0,C 180,E1 -25894.417,E2 -25894.417} C_VEL
LIN {X 0,Y 127.679,Z 290.684,A -85,B 0,C 180,E1 -25899.037,E2 -25899.037} C_VEL
LIN {X 0,Y 125.56,Z 287.961,A -85,B 0,C 180,E1 -25903.33,E2 -25903.33} C_VEL
LIN {X 0,Y 124.83,Z 285.838,A -85,B 0,C 180,E1 -25905.74,E2 -25905.74} C_VEL
LIN {X 0,Y 122.287,Z 282.577,A -85,B 0,C 180,E1 -25920,E2 -25920} C_VEL
LIN {X 0,Y 123.453,Z 286.509,A -85,B 0,C 180,E1 -25929.833,E2 -25929.833} C_VEL
LIN {X 0,Y 125.488,Z 289.224,A -85,B 0,C 180,E1 -25935.22,E2 -25935.22} C_VEL
LIN {X 0,Y 126.871,Z 293.06,A -85,B 0,C 180,E1 -25938.783,E2 -25938.783} C_VEL
LIN {X 0,Y 128.485,Z 295.433,A -85,B 0,C 180,E1 -25941.584,E2 -25941.584} C_VEL
LIN {X 0,Y 129.647,Z 298.797,A -85,B 0,C 180,E1 -25943.989,E2 -25943.989} C_VEL
LIN {X 0,Y 131.136,Z 301.659,A -85,B 0,C 180,E1 -25946.346,E2 -25946.346} C_VEL
LIN {X 0,Y 133.345,Z 307.35,A -85,B 0,C 180,E1 -25950.046,E2 -25950.046} C_VEL
LIN {X 0,Y 135.724,Z 314.313,A -85,B 0,C 180,E1 -25954.055,E2 -25954.055} C_VEL
LIN {X 0,Y 137.716,Z 321.507,A -85,B 0,C 180,E1 -25957.762,E2 -25957.762} C_VEL
LIN {X 0,Y 138.489,Z 326.191,A -85,B 0,C 180,E1 -25959.927,E2 -25959.927} C_VEL
LIN {X 0,Y 137.219,Z 336.185,A -85,B 0,C 180,E1 -25963.547,E2 -25963.547} C_VEL
LIN {X 0,Y 134.951,Z 345.969,A -85,B 0,C 180,E1 -25967.389,E2 -25967.389} C_VEL
LIN {X 0,Y 132.633,Z 353.01,A -85,B 0,C 180,E1 -25970.517,E2 -25970.517} C_VEL
LIN {X 0,Y 130.332,Z 357.623,A -85,B 0,C 180,E1 -25972.653,E2 -25972.653} C_VEL
LIN {X 0,Y 125.207,Z 365.455,A -85,B 0,C 180,E1 -25976.916,E2 -25976.916} C_VEL
LIN {X 0,Y 121.86,Z 370.659,A -85,B 0,C 180,E1 -25980.645,E2 -25980.645} C_VEL
LIN {X 0,Y 118.242,Z 375.807,A -85,B 0,C 180,E1 -25985.414,E2 -25985.414} C_VEL
LIN {X 0,Y 115.419,Z 379.816,A -85,B 0,C 180,E1 -25990.434,E2 -25990.434} C_VEL
LIN {X 0,Y 113.624,Z 382.801,A -85,B 0,C 180,E1 -25995.676,E2 -25995.676} C_VEL
LIN {X 0,Y 112.571,Z 385.261,A -85,B 0,C 180,E1 -26002.828,E2 -26002.828} C_VEL
LIN {X 0,Y 112.546,Z 386.015,A -85,B 0,C 180,E1 -26007.604,E2 -26007.604} C_VEL
LIN {X 0,Y 112.696,Z 386.128,A -85,B 0,C 180,E1 -26010.001,E2 -26010.001} C_VEL
LIN {X 0,Y 112.517,Z 385.882,A -85,B 0,C 180,E1 -26013.582,E2 -26013.582} C_VEL
LIN {X 0,Y 112.571,Z 385.238,A -85,B 0,C 180,E1 -26017.173,E2 -26017.173} C_VEL
LIN {X 0,Y 112.904,Z 384.198,A -85,B 0,C 180,E1 -26020.763,E2 -26020.763} C_VEL
LIN {X 0,Y 113.623,Z 382.754,A -85,B 0,C 180,E1 -26024.325,E2 -26024.325} C_VEL
LIN {X 0,Y 115.418,Z 379.749,A -85,B 0,C 180,E1 -26029.567,E2 -26029.567} C_VEL
LIN {X 0,Y 118.235,Z 375.715,A -85,B 0,C 180,E1 -26034.589,E2 -26034.589} C_VEL
LIN {X 0,Y 122.465,Z 369.524,A -85,B 0,C 180,E1 -26040.143,E2 -26040.143} C_VEL
LIN {X 0,Y 126.885,Z 362.779,A -85,B 0,C 180,E1 -26044.593,E2 -26044.593} C_VEL
LIN {X 0,Y 131.196,Z 355.935,A -85,B 0,C 180,E1 -26048.029,E2 -26048.029} C_VEL
LIN {X 0,Y 133.796,Z 349.402,A -85,B 0,C 180,E1 -26051.042,E2 -26051.042} C_VEL
LIN {X 0,Y 135.959,Z 341.517,A -85,B 0,C 180,E1 -26054.345,E2 -26054.345} C_VEL
LIN {X 0,Y 137.866,Z 331.523,A -85,B 0,C 180,E1 -26058.061,E2 -26058.061} C_VEL
LIN {X 0,Y 138.413,Z 325.807,A -85,B 0,C 180,E1 -26060.109,E2 -26060.109} C_VEL
LIN {X 0,Y 137.205,Z 319.711,A -85,B 0,C 180,E1 -26062.996,E2 -26062.996} C_VEL
LIN {X 0,Y 134.665,Z 311.082,A -85,B 0,C 180,E1 -26067.572,E2 -26067.572} C_VEL
LIN {X 0,Y 132.257,Z 304.79,A -85,B 0,C 180,E1 -26071.429,E2 -26071.429} C_VEL
LIN {X 0,Y 130.459,Z 300.316,A -85,B 0,C 180,E1 -26074.471,E2 -26074.471} C_VEL
LIN {X 0,Y 128.724,Z 296.283,A -85,B 0,C 180,E1 -26077.531,E2 -26077.531} C_VEL
LIN {X 0,Y 125.644,Z 290.183,A -85,B 0,C 180,E1 -26083.655,E2 -26083.655} C_VEL
LIN {X 0,Y 125.387,Z 289.035,A -85,B 0,C 180,E1 -26084.559,E2 -26084.559} C_VEL
LIN {X 0,Y 122.125,Z 283.497,A -85,B 0,C 180,E1 -26096.288,E2 -26096.288} C_VEL
LIN {X 0,Y 122.08,Z 282.128,A -85,B 0,C 180,E1 -26100,E2 -26100} C_VEL
LIN {X 0,Y 123.594,Z 285.061,A -85,B 0,C 180,E1 -26111.844,E2 -26111.844} C_VEL
LIN {X 0,Y 123.981,Z 286.35,A -85,B 0,C 180,E1 -26113.55,E2 -26113.55} C_VEL
LIN {X 0,Y 124.04,Z 289.563,A -85,B 0,C 180,E1 -26115.532,E2 -26115.532} C_VEL
LIN {X 0,Y 123.888,Z 294.937,A -85,B 0,C 180,E1 -26118.417,E2 -26118.417} C_VEL
LIN {X 0,Y 124.324,Z 296.717,A -85,B 0,C 180,E1 -26120.083,E2 -26120.083} C_VEL
LIN {X 0,Y 124.998,Z 297.596,A -85,B 0,C 180,E1 -26121.436,E2 -26121.436} C_VEL
LIN {X 0,Y 127.275,Z 302.055,A -85,B 0,C 180,E1 -26126.216,E2 -26126.216} C_VEL
LIN {X 0,Y 129.342,Z 306.47,A -85,B 0,C 180,E1 -26130.173,E2 -26130.173} C_VEL
LIN {X 0,Y 131.697,Z 312.289,A -85,B 0,C 180,E1 -26134.633,E2 -26134.633} C_VEL
LIN {X 0,Y 133.367,Z 317.7,A -85,B 0,C 180,E1 -26138.257,E2 -26138.257} C_VEL
LIN {X 0,Y 134.266,Z 322.53,A -85,B 0,C 180,E1 -26141.133,E2 -26141.133} C_VEL
LIN {X 0,Y 134.403,Z 328.483,A -85,B 0,C 180,E1 -26144.287,E2 -26144.287} C_VEL
LIN {X 0,Y 133.887,Z 334.324,A -85,B 0,C 180,E1 -26147.298,E2 -26147.298} C_VEL
LIN {X 0,Y 130.451,Z 340.563,A -85,B 0,C 180,E1 -26149.721,E2 -26149.721} C_VEL
LIN {X 0,Y 124.847,Z 349.131,A -85,B 0,C 180,E1 -26153.766,E2 -26153.766} C_VEL
LIN {X 0,Y 119.851,Z 355.957,A -85,B 0,C 180,E1 -26158.145,E2 -26158.145} C_VEL
LIN {X 0,Y 115.518,Z 361.419,A -85,B 0,C 180,E1 -26162.851,E2 -26162.851} C_VEL
LIN {X 0,Y 111.961,Z 365.697,A -85,B 0,C 180,E1 -26167.874,E2 -26167.874} C_VEL
LIN {X 0,Y 110.038,Z 367.958,A -85,B 0,C 180,E1 -26171.376,E2 -26171.376} C_VEL
LIN {X 0,Y 108.555,Z 369.788,A -85,B 0,C 180,E1 -26174.991,E2 -26174.991} C_VEL
LIN {X 0,Y 107.209,Z 371.407,A -85,B 0,C 180,E1 -26179.519,E2 -26179.519} C_VEL
LIN {X 0,Y 106.056,Z 372.739,A -85,B 0,C 180,E1 -26186.2,E2 -26186.2} C_VEL
LIN {X 0,Y 105.888,Z 372.962,A -85,B 0,C 180,E1 -26189.999,E2 -26189.999} C_VEL
LIN {X 0,Y 106.052,Z 372.766,A -85,B 0,C 180,E1 -26193.799,E2 -26193.799} C_VEL
LIN {X 0,Y 107.361,Z 371.224,A -85,B 0,C 180,E1 -26201.325,E2 -26201.325} C_VEL
LIN {X 0,Y 108.515,Z 369.878,A -85,B 0,C 180,E1 -26205.014,E2 -26205.014} C_VEL
LIN {X 0,Y 110.934,Z 367.03,A -85,B 0,C 180,E1 -26210.392,E2 -26210.392} C_VEL
LIN {X 0,Y 114.198,Z 363.16,A -85,B 0,C 180,E1 -26215.518,E2 -26215.518} C_VEL
LIN {X 0,Y 118.246,Z 358.162,A -85,B 0,C 180,E1 -26220.344,E2 -26220.344} C_VEL
LIN {X 0,Y 122.987,Z 351.858,A -85,B 0,C 180,E1 -26224.85,E2 -26224.85} C_VEL
LIN {X 0,Y 128.456,Z 343.961,A -85,B 0,C 180,E1 -26228.99,E2 -26228.99} C_VEL
LIN {X 0,Y 133.011,Z 336.445,A -85,B 0,C 180,E1 -26232.045,E2 -26232.045} C_VEL
LIN {X 0,Y 134.024,Z 334.169,A -85,B 0,C 180,E1 -26232.976,E2 -26232.976} C_VEL
LIN {X 0,Y 134.566,Z 326.429,A -85,B 0,C 180,E1 -26236.985,E2 -26236.985} C_VEL
LIN {X 0,Y 134.114,Z 321.231,A -85,B 0,C 180,E1 -26239.873,E2 -26239.873} C_VEL
LIN {X 0,Y 133.321,Z 317.289,A -85,B 0,C 180,E1 -26242.253,E2 -26242.253} C_VEL
LIN {X 0,Y 131.482,Z 311.707,A -85,B 0,C 180,E1 -26246.08,E2 -26246.08} C_VEL
LIN {X 0,Y 129.157,Z 305.721,A -85,B 0,C 180,E1 -26250.677,E2 -26250.677} C_VEL
LIN {X 0,Y 126.649,Z 300.875,A -85,B 0,C 180,E1 -26255.405,E2 -26255.405} C_VEL
LIN {X 0,Y 124.472,Z 296.761,A -85,B 0,C 180,E1 -26260.198,E2 -26260.198} C_VEL
LIN {X 0,Y 123.139,Z 294.84,A -85,B 0,C 180,E1 -26263.419,E2 -26263.419} C_VEL
LIN {X 0,Y 122.283,Z 292.373,A -85,B 0,C 180,E1 -26266.709,E2 -26266.709} C_VEL
LIN {X 0,Y 120.44,Z 289.531,A -85,B 0,C 180,E1 -26280,E2 -26280} C_VEL
LIN {X 0,Y 120.783,Z 292.002,A -85,B 0,C 180,E1 -26286.683,E2 -26286.683} C_VEL
LIN {X 0,Y 122.504,Z 295.017,A -85,B 0,C 180,E1 -26293.266,E2 -26293.266} C_VEL
LIN {X 0,Y 125.255,Z 301.378,A -85,B 0,C 180,E1 -26300.535,E2 -26300.535} C_VEL
LIN {X 0,Y 127.709,Z 308.444,A -85,B 0,C 180,E1 -26306.12,E2 -26306.12} C_VEL
LIN {X 0,Y 129.378,Z 313.599,A -85,B 0,C 180,E1 -26309.641,E2 -26309.641} C_VEL
LIN {X 0,Y 130.769,Z 318.141,A -85,B 0,C 180,E1 -26312.509,E2 -26312.509} C_VEL
LIN {X 0,Y 132.457,Z 325.494,A -85,B 0,C 180,E1 -26316.649,E2 -26316.649} C_VEL
LIN {X 0,Y 132.941,Z 328.765,A -85,B 0,C 180,E1 -26318.341,E2 -26318.341} C_VEL
LIN {X 0,Y 131.84,Z 335.781,A -85,B 0,C 180,E1 -26321.063,E2 -26321.063} C_VEL
LIN {X 0,Y 129.932,Z 343.718,A -85,B 0,C 180,E1 -26324.33,E2 -26324.33} C_VEL
LIN {X 0,Y 127.625,Z 350.896,A -85,B 0,C 180,E1 -26327.579,E2 -26327.579} C_VEL
LIN {X 0,Y 125.599,Z 355.695,A -85,B 0,C 180,E1 -26329.948,E2 -26329.948} C_VEL
LIN {X 0,Y 120.215,Z 363.752,A -85,B 0,C 180,E1 -26334.224,E2 -26334.224} C_VEL
LIN {X 0,Y 115.637,Z 370.227,A -85,B 0,C 180,E1 -26338.896,E2 -26338.896} C_VEL
LIN {X 0,Y 111.77,Z 375.377,A -85,B 0,C 180,E1 -26343.887,E2 -26343.887} C_VEL
LIN {X 0,Y 108.733,Z 379.388,A -85,B 0,C 180,E1 -26349.177,E2 -26349.177} C_VEL
LIN {X 0,Y 106.72,Z 382.372,A -85,B 0,C 180,E1 -26354.727,E2 -26354.727} C_VEL
LIN {X 0,Y 105.505,Z 384.832,A -85,B 0,C 180,E1 -26362.344,E2 -26362.344} C_VEL
LIN {X 0,Y 105.478,Z 385.619,A -85,B 0,C 180,E1 -26368.093,E2 -26368.093} C_VEL
LIN {X 0,Y 105.476,Z 385.615,A -85,B 0,C 180,E1 -26371.871,E2 -26371.871} C_VEL
LIN {X 0,Y 105.505,Z 384.808,A -85,B 0,C 180,E1 -26377.657,E2 -26377.657} C_VEL
LIN {X 0,Y 106.719,Z 382.324,A -85,B 0,C 180,E1 -26385.274,E2 -26385.274} C_VEL
LIN {X 0,Y 108.732,Z 379.319,A -85,B 0,C 180,E1 -26390.825,E2 -26390.825} C_VEL
LIN {X 0,Y 111.763,Z 375.283,A -85,B 0,C 180,E1 -26396.116,E2 -26396.116} C_VEL
LIN {X 0,Y 115.651,Z 370.105,A -85,B 0,C 180,E1 -26401.101,E2 -26401.101} C_VEL
LIN {X 0,Y 121.079,Z 362.347,A -85,B 0,C 180,E1 -26406.511,E2 -26406.511} C_VEL
LIN {X 0,Y 125.562,Z 355.496,A -85,B 0,C 180,E1 -26410.068,E2 -26410.068} C_VEL
LIN {X 0,Y 128.228,Z 348.947,A -85,B 0,C 180,E1 -26413.245,E2 -26413.245} C_VEL
LIN {X 0,Y 131.034,Z 339.044,A -85,B 0,C 180,E1 -26417.517,E2 -26417.517} C_VEL
LIN {X 0,Y 132.793,Z 329.787,A -85,B 0,C 180,E1 -26421.117,E2 -26421.117} C_VEL
LIN {X 0,Y 132.596,Z 326.559,A -85,B 0,C 180,E1 -26422.661,E2 -26422.661} C_VEL
LIN {X 0,Y 130.653,Z 317.937,A -85,B 0,C 180,E1 -26427.458,E2 -26427.458} C_VEL
LIN {X 0,Y 128.367,Z 310.423,A -85,B 0,C 180,E1 -26432.266,E2 -26432.266} C_VEL
LIN {X 0,Y 126.845,Z 306.023,A -85,B 0,C 180,E1 -26435.446,E2 -26435.446} C_VEL
LIN {X 0,Y 125.282,Z 301.846,A -85,B 0,C 180,E1 -26438.878,E2 -26438.878} C_VEL
LIN {X 0,Y 123.3,Z 297.687,A -85,B 0,C 180,E1 -26443.441,E2 -26443.441} C_VEL
LIN {X 0,Y 122.848,Z 295.929,A -85,B 0,C 180,E1 -26445.082,E2 -26445.082} C_VEL
LIN {X 0,Y 121.242,Z 293.246,A -85,B 0,C 180,E1 -26449.985,E2 -26449.985} C_VEL
LIN {X 0,Y 120.208,Z 289.505,A -85,B 0,C 180,E1 -26458.744,E2 -26458.744} C_VEL
LIN {X 0,Y 120.258,Z 289.068,A -85,B 0,C 180,E1 -26460,E2 -26460} C_VEL
LIN {X 0,Y 121.974,Z 292.307,A -85,B 0,C 180,E1 -26473.325,E2 -26473.325} C_VEL
LIN {X 0,Y 122.52,Z 293.045,A -85,B 0,C 180,E1 -26474.959,E2 -26474.959} C_VEL
LIN {X 0,Y 123.336,Z 295.371,A -85,B 0,C 180,E1 -26477.84,E2 -26477.84} C_VEL
LIN {X 0,Y 124.324,Z 296.717,A -85,B 0,C 180,E1 -26480.083,E2 -26480.083} C_VEL
LIN {X 0,Y 125.256,Z 299.094,A -85,B 0,C 180,E1 -26482.516,E2 -26482.516} C_VEL
LIN {X 0,Y 125.635,Z 302.475,A -85,B 0,C 180,E1 -26484.744,E2 -26484.744} C_VEL
LIN {X 0,Y 125.789,Z 312.785,A -85,B 0,C 180,E1 -26490.429,E2 -26490.429} C_VEL
LIN {X 0,Y 126.186,Z 314.96,A -85,B 0,C 180,E1 -26491.973,E2 -26491.973} C_VEL
LIN {X 0,Y 127.824,Z 320.504,A -85,B 0,C 180,E1 -26496.231,E2 -26496.231} C_VEL
LIN {X 0,Y 128.774,Z 326.478,A -85,B 0,C 180,E1 -26500.175,E2 -26500.175} C_VEL
LIN {X 0,Y 128.482,Z 332.946,A -85,B 0,C 180,E1 -26503.9,E2 -26503.9} C_VEL
LIN {X 0,Y 128.034,Z 335.87,A -85,B 0,C 180,E1 -26505.528,E2 -26505.528} C_VEL
LIN {X 0,Y 126.5,Z 338.861,A -85,B 0,C 180,E1 -26506.761,E2 -26506.761} C_VEL
LIN {X 0,Y 121.092,Z 346.9,A -85,B 0,C 180,E1 -26510.325,E2 -26510.325} C_VEL
LIN {X 0,Y 115.572,Z 354.265,A -85,B 0,C 180,E1 -26514.71,E2 -26514.71} C_VEL
LIN {X 0,Y 110.72,Z 360.168,A -85,B 0,C 180,E1 -26519.481,E2 -26519.481} C_VEL
LIN {X 0,Y 106.627,Z 364.827,A -85,B 0,C 180,E1 -26524.631,E2 -26524.631} C_VEL
LIN {X 0,Y 103.35,Z 368.385,A -85,B 0,C 180,E1 -26530.122,E2 -26530.122} C_VEL
LIN {X 0,Y 101.736,Z 370.215,A -85,B 0,C 180,E1 -26533.958,E2 -26533.958} C_VEL
LIN {X 0,Y 100.092,Z 372.012,A -85,B 0,C 180,E1 -26539.428,E2 -26539.428} C_VEL
LIN {X 0,Y 99.002,Z 373.165,A -85,B 0,C 180,E1 -26545.929,E2 -26545.929} C_VEL
LIN {X 0,Y 98.818,Z 373.388,A -85,B 0,C 180,E1 -26549.999,E2 -26549.999} C_VEL
LIN {X 0,Y 98.998,Z 373.192,A -85,B 0,C 180,E1 -26554.07,E2 -26554.07} C_VEL
LIN {X 0,Y 100.425,Z 371.65,A -85,B 0,C 180,E1 -26562.119,E2 -26562.119} C_VEL
LIN {X 0,Y 101.685,Z 370.304,A -85,B 0,C 180,E1 -26566.049,E2 -26566.049} C_VEL
LIN {X 0,Y 104.327,Z 367.456,A -85,B 0,C 180,E1 -26571.747,E2 -26571.747} C_VEL
LIN {X 0,Y 107.834,Z 363.587,A -85,B 0,C 180,E1 -26577.143,E2 -26577.143} C_VEL
LIN {X 0,Y 112.196,Z 358.586,A -85,B 0,C 180,E1 -26582.17,E2 -26582.17} C_VEL
LIN {X 0,Y 117.254,Z 352.281,A -85,B 0,C 180,E1 -26586.825,E2 -26586.825} C_VEL
LIN {X 0,Y 123.033,Z 344.385,A -85,B 0,C 180,E1 -26591.065,E2 -26591.065} C_VEL
LIN {X 0,Y 127.221,Z 337.923,A -85,B 0,C 180,E1 -26593.784,E2 -26593.784} C_VEL
LIN {X 0,Y 128.097,Z 336.173,A -85,B 0,C 180,E1 -26594.5,E2 -26594.5} C_VEL
LIN {X 0,Y 128.87,Z 329.54,A -85,B 0,C 180,E1 -26598.239,E2 -26598.239} C_VEL
LIN {X 0,Y 128.733,Z 325.545,A -85,B 0,C 180,E1 -26600.655,E2 -26600.655} C_VEL
LIN {X 0,Y 127.968,Z 320.793,A -85,B 0,C 180,E1 -26603.816,E2 -26603.816} C_VEL
LIN {X 0,Y 126.009,Z 314.201,A -85,B 0,C 180,E1 -26608.941,E2 -26608.941} C_VEL
LIN {X 0,Y 125.003,Z 311.261,A -85,B 0,C 180,E1 -26611.452,E2 -26611.452} C_VEL
LIN {X 0,Y 122.896,Z 306.534,A -85,B 0,C 180,E1 -26616.402,E2 -26616.402} C_VEL
LIN {X 0,Y 121.712,Z 303.726,A -85,B 0,C 180,E1 -26619.729,E2 -26619.729} C_VEL
LIN {X 0,Y 119.75,Z 299.412,A -85,B 0,C 180,E1 -26626.423,E2 -26626.423} C_VEL
LIN {X 0,Y 118.306,Z 297.508,A -85,B 0,C 180,E1 -26633.176,E2 -26633.176} C_VEL
LIN {X 0,Y 118.223,Z 296.351,A -85,B 0,C 180,E1 -26640,E2 -26640} C_VEL
LIN {X 0,Y 119.063,Z 300.322,A -85,B 0,C 180,E1 -26650.2,E2 -26650.2} C_VEL
LIN {X 0,Y 119.971,Z 302.152,A -85,B 0,C 180,E1 -26653.552,E2 -26653.552} C_VEL
LIN {X 0,Y 121.973,Z 308.096,A -85,B 0,C 180,E1 -26660.225,E2 -26660.225} C_VEL
LIN {X 0,Y 123.714,Z 313.978,A -85,B 0,C 180,E1 -26665.216,E2 -26665.216} C_VEL
LIN {X 0,Y 125.584,Z 320.929,A -85,B 0,C 180,E1 -26670.242,E2 -26670.242} C_VEL
LIN {X 0,Y 126.892,Z 327.861,A -85,B 0,C 180,E1 -26674.59,E2 -26674.59} C_VEL
LIN {X 0,Y 127.322,Z 330.977,A -85,B 0,C 180,E1 -26676.398,E2 -26676.398} C_VEL
LIN {X 0,Y 127.02,Z 334.283,A -85,B 0,C 180,E1 -26677.959,E2 -26677.959} C_VEL
LIN {X 0,Y 124.716,Z 343.053,A -85,B 0,C 180,E1 -26681.698,E2 -26681.698} C_VEL
LIN {X 0,Y 122.11,Z 350.624,A -85,B 0,C 180,E1 -26685.291,E2 -26685.291} C_VEL
LIN {X 0,Y 119.252,Z 356.765,A -85,B 0,C 180,E1 -26688.471,E2 -26688.471} C_VEL
LIN {X 0,Y 113.607,Z 364.486,A -85,B 0,C 180,E1 -26692.904,E2 -26692.904} C_VEL
LIN {X 0,Y 109.387,Z 370.008,A -85,B 0,C 180,E1 -26697.151,E2 -26697.151} C_VEL
LIN {X 0,Y 105.392,Z 374.947,A -85,B 0,C 180,E1 -26702.174,E2 -26702.174} C_VEL
LIN {X 0,Y 102.085,Z 378.958,A -85,B 0,C 180,E1 -26707.751,E2 -26707.751} C_VEL
LIN {X 0,Y 99.833,Z 381.941,A -85,B 0,C 180,E1 -26713.645,E2 -26713.645} C_VEL
LIN {X 0,Y 98.449,Z 384.403,A -85,B 0,C 180,E1 -26721.792,E2 -26721.792} C_VEL
LIN {X 0,Y 98.43,Z 385.214,A -85,B 0,C 180,E1 -26728.417,E2 -26728.417} C_VEL
LIN {X 0,Y 98.419,Z 385.218,A -85,B 0,C 180,E1 -26731.336,E2 -26731.336} C_VEL
LIN {X 0,Y 98.449,Z 384.379,A -85,B 0,C 180,E1 -26738.209,E2 -26738.209} C_VEL
LIN {X 0,Y 98.922,Z 383.338,A -85,B 0,C 180,E1 -26742.307,E2 -26742.307} C_VEL
LIN {X 0,Y 99.833,Z 381.892,A -85,B 0,C 180,E1 -26746.356,E2 -26746.356} C_VEL
LIN {X 0,Y 102.084,Z 378.888,A -85,B 0,C 180,E1 -26752.251,E2 -26752.251} C_VEL
LIN {X 0,Y 105.386,Z 374.85,A -85,B 0,C 180,E1 -26757.829,E2 -26757.829} C_VEL
LIN {X 0,Y 109.132,Z 370.244,A -85,B 0,C 180,E1 -26762.514,E2 -26762.514} C_VEL
LIN {X 0,Y 114.496,Z 363.159,A -85,B 0,C 180,E1 -26767.867,E2 -26767.867} C_VEL
LIN {X 0,Y 119.219,Z 356.565,A -85,B 0,C 180,E1 -26771.545,E2 -26771.545} C_VEL
LIN {X 0,Y 122.063,Z 350.422,A -85,B 0,C 180,E1 -26774.716,E2 -26774.716} C_VEL
LIN {X 0,Y 125.293,Z 340.759,A -85,B 0,C 180,E1 -26779.224,E2 -26779.224} C_VEL
LIN {X 0,Y 127.212,Z 332.733,A -85,B 0,C 180,E1 -26782.576,E2 -26782.576} C_VEL
LIN {X 0,Y 127.044,Z 329.14,A -85,B 0,C 180,E1 -26784.489,E2 -26784.489} C_VEL
LIN {X 0,Y 125.738,Z 322.043,A -85,B 0,C 180,E1 -26788.866,E2 -26788.866} C_VEL
LIN {X 0,Y 124.247,Z 315.892,A -85,B 0,C 180,E1 -26793.095,E2 -26793.095} C_VEL
LIN {X 0,Y 123.001,Z 311.6,A -85,B 0,C 180,E1 -26796.424,E2 -26796.424} C_VEL
LIN {X 0,Y 121.822,Z 307.831,A -85,B 0,C 180,E1 -26799.748,E2 -26799.748} C_VEL
LIN {X 0,Y 119.805,Z 301.841,A -85,B 0,C 180,E1 -26806.429,E2 -26806.429} C_VEL
LIN {X 0,Y 117.994,Z 297.128,A -85,B 0,C 180,E1 -26816.585,E2 -26816.585} C_VEL
LIN {X 0,Y 118.053,Z 295.922,A -85,B 0,C 180,E1 -26820,E2 -26820} C_VEL
LIN {X 0,Y 118.614,Z 298.146,A -85,B 0,C 180,E1 -26830.239,E2 -26830.239} C_VEL
LIN {X 0,Y 119.523,Z 299.14,A -85,B 0,C 180,E1 -26833.604,E2 -26833.604} C_VEL
LIN {X 0,Y 121.503,Z 303.44,A -85,B 0,C 180,E1 -26840.307,E2 -26840.307} C_VEL
LIN {X 0,Y 123.413,Z 307.678,A -85,B 0,C 180,E1 -26845.284,E2 -26845.284} C_VEL
LIN {X 0,Y 125.502,Z 312.931,A -85,B 0,C 180,E1 -26850.265,E2 -26850.265} C_VEL
LIN {X 0,Y 126.186,Z 314.96,A -85,B 0,C 180,E1 -26851.973,E2 -26851.973} C_VEL
LIN {X 0,Y 126.607,Z 318.369,A -85,B 0,C 180,E1 -26854.176,E2 -26854.176} C_VEL
LIN {X 0,Y 125.864,Z 323.818,A -85,B 0,C 180,E1 -26856.817,E2 -26856.817} C_VEL
LIN {X 0,Y 123.955,Z 330.907,A -85,B 0,C 180,E1 -26860.028,E2 -26860.028} C_VEL
LIN {X 0,Y 122.568,Z 336.158,A -85,B 0,C 180,E1 -26862.827,E2 -26862.827} C_VEL
LIN {X 0,Y 122.318,Z 337.412,A -85,B 0,C 180,E1 -26863.589,E2 -26863.589} C_VEL
LIN {X 0,Y 121.56,Z 339.12,A -85,B 0,C 180,E1 -26864.406,E2 -26864.406} C_VEL
LIN {X 0,Y 115.734,Z 347.329,A -85,B 0,C 180,E1 -26868.088,E2 -26868.088} C_VEL
LIN {X 0,Y 109.866,Z 354.693,A -85,B 0,C 180,E1 -26872.575,E2 -26872.575} C_VEL
LIN {X 0,Y 104.677,Z 360.596,A -85,B 0,C 180,E1 -26877.512,E2 -26877.512} C_VEL
LIN {X 0,Y 100.269,Z 365.255,A -85,B 0,C 180,E1 -26882.896,E2 -26882.896} C_VEL
LIN {X 0,Y 96.728,Z 368.812,A -85,B 0,C 180,E1 -26888.697,E2 -26888.697} C_VEL
LIN {X 0,Y 94.943,Z 370.642,A -85,B 0,C 180,E1 -26892.776,E2 -26892.776} C_VEL
LIN {X 0,Y 92.892,Z 372.683,A -85,B 0,C 180,E1 -26899.595,E2 -26899.595} C_VEL
LIN {X 0,Y 91.933,Z 373.592,A -85,B 0,C 180,E1 -26905.615,E2 -26905.615} C_VEL
LIN {X 0,Y 91.749,Z 373.814,A -85,B 0,C 180,E1 -26909.999,E2 -26909.999} C_VEL
LIN {X 0,Y 91.928,Z 373.618,A -85,B 0,C 180,E1 -26914.384,E2 -26914.384} C_VEL
LIN {X 0,Y 93.513,Z 372.076,A -85,B 0,C 180,E1 -26923.03,E2 -26923.03} C_VEL
LIN {X 0,Y 94.883,Z 370.731,A -85,B 0,C 180,E1 -26927.234,E2 -26927.234} C_VEL
LIN {X 0,Y 97.79,Z 367.881,A -85,B 0,C 180,E1 -26933.283,E2 -26933.283} C_VEL
LIN {X 0,Y 101.576,Z 364.013,A -85,B 0,C 180,E1 -26938.968,E2 -26938.968} C_VEL
LIN {X 0,Y 106.273,Z 359.011,A -85,B 0,C 180,E1 -26944.202,E2 -26944.202} C_VEL
LIN {X 0,Y 111.674,Z 352.705,A -85,B 0,C 180,E1 -26949.001,E2 -26949.001} C_VEL
LIN {X 0,Y 117.789,Z 344.808,A -85,B 0,C 180,E1 -26953.327,E2 -26953.327} C_VEL
LIN {X 0,Y 121.511,Z 339.419,A -85,B 0,C 180,E1 -26955.664,E2 -26955.664} C_VEL
LIN {X 0,Y 122.366,Z 337.733,A -85,B 0,C 180,E1 -26956.432,E2 -26956.432} C_VEL
LIN {X 0,Y 123.161,Z 332.88,A -85,B 0,C 180,E1 -26959.394,E2 -26959.394} C_VEL
LIN {X 0,Y 123.178,Z 328.743,A -85,B 0,C 180,E1 -26962.168,E2 -26962.168} C_VEL
LIN {X 0,Y 122.538,Z 323.905,A -85,B 0,C 180,E1 -26965.802,E2 -26965.802} C_VEL
LIN {X 0,Y 121.206,Z 318.588,A -85,B 0,C 180,E1 -26970.43,E2 -26970.43} C_VEL
LIN {X 0,Y 120.038,Z 315.093,A -85,B 0,C 180,E1 -26973.952,E2 -26973.952} C_VEL
LIN {X 0,Y 118.946,Z 312.062,A -85,B 0,C 180,E1 -26977.415,E2 -26977.415} C_VEL
LIN {X 0,Y 118.014,Z 309.401,A -85,B 0,C 180,E1 -26980.88,E2 -26980.88} C_VEL
LIN {X 0,Y 116.748,Z 306.393,A -85,B 0,C 180,E1 -26986.066,E2 -26986.066} C_VEL
LIN {X 0,Y 116.119,Z 304.942,A -85,B 0,C 180,E1 -26989.538,E2 -26989.538} C_VEL
LIN {X 0,Y 115.419,Z 303.478,A -85,B 0,C 180,E1 -26996.509,E2 -26996.509} C_VEL
LIN {X 0,Y 115.58,Z 303.046,A -85,B 0,C 180,E1 -27000,E2 -27000} C_VEL
LIN {X 0,Y 115.692,Z 305.564,A -85,B 0,C 180,E1 -27006.978,E2 -27006.978} C_VEL
LIN {X 0,Y 116.661,Z 307.989,A -85,B 0,C 180,E1 -27012.172,E2 -27012.172} C_VEL
LIN {X 0,Y 118.185,Z 313.627,A -85,B 0,C 180,E1 -27019.091,E2 -27019.091} C_VEL
LIN {X 0,Y 119.502,Z 319.357,A -85,B 0,C 180,E1 -27024.31,E2 -27024.31} C_VEL
LIN {X 0,Y 120.779,Z 325.663,A -85,B 0,C 180,E1 -27029.211,E2 -27029.211} C_VEL
LIN {X 0,Y 121.653,Z 332.558,A -85,B 0,C 180,E1 -27033.894,E2 -27033.894} C_VEL
LIN {X 0,Y 121.799,Z 334.711,A -85,B 0,C 180,E1 -27035.241,E2 -27035.241} C_VEL
LIN {X 0,Y 121.144,Z 337.841,A -85,B 0,C 180,E1 -27036.745,E2 -27036.745} C_VEL
LIN {X 0,Y 118.291,Z 346.514,A -85,B 0,C 180,E1 -27040.809,E2 -27040.809} C_VEL
LIN {X 0,Y 115.459,Z 353.285,A -85,B 0,C 180,E1 -27044.339,E2 -27044.339} C_VEL
LIN {X 0,Y 112.97,Z 357.719,A -85,B 0,C 180,E1 -27046.818,E2 -27046.818} C_VEL
LIN {X 0,Y 107.063,Z 365.187,A -85,B 0,C 180,E1 -27051.42,E2 -27051.42} C_VEL
LIN {X 0,Y 102.083,Z 371.208,A -85,B 0,C 180,E1 -27056.581,E2 -27056.581} C_VEL
LIN {X 0,Y 97.838,Z 375.969,A -85,B 0,C 180,E1 -27062.166,E2 -27062.166} C_VEL
LIN {X 0,Y 94.521,Z 379.617,A -85,B 0,C 180,E1 -27068.176,E2 -27068.176} C_VEL
LIN {X 0,Y 92.999,Z 381.512,A -85,B 0,C 180,E1 -27072.406,E2 -27072.406} C_VEL
LIN {X 0,Y 91.391,Z 383.974,A -85,B 0,C 180,E1 -27081.153,E2 -27081.153} C_VEL
LIN {X 0,Y 91.378,Z 384.816,A -85,B 0,C 180,E1 -27089.01,E2 -27089.01} C_VEL
LIN {X 0,Y 91.23,Z 384.596,A -85,B 0,C 180,E1 -27094.419,E2 -27094.419} C_VEL
LIN {X 0,Y 91.391,Z 383.948,A -85,B 0,C 180,E1 -27098.848,E2 -27098.848} C_VEL
LIN {X 0,Y 91.952,Z 382.907,A -85,B 0,C 180,E1 -27103.256,E2 -27103.256} C_VEL
LIN {X 0,Y 92.999,Z 381.461,A -85,B 0,C 180,E1 -27107.596,E2 -27107.596} C_VEL
LIN {X 0,Y 95.516,Z 378.457,A -85,B 0,C 180,E1 -27113.872,E2 -27113.872} C_VEL
LIN {X 0,Y 99.12,Z 374.419,A -85,B 0,C 180,E1 -27119.758,E2 -27119.758} C_VEL
LIN {X 0,Y 103.745,Z 369.034,A -85,B 0,C 180,E1 -27125.4,E2 -27125.4} C_VEL
LIN {X 0,Y 108.95,Z 362.727,A -85,B 0,C 180,E1 -27130.172,E2 -27130.172} C_VEL
LIN {X 0,Y 113.852,Z 356.122,A -85,B 0,C 180,E1 -27133.985,E2 -27133.985} C_VEL
LIN {X 0,Y 117.188,Z 349.042,A -85,B 0,C 180,E1 -27137.824,E2 -27137.824} C_VEL
LIN {X 0,Y 120.356,Z 340.286,A -85,B 0,C 180,E1 -27142.03,E2 -27142.03} C_VEL
LIN {X 0,Y 121.583,Z 335.865,A -85,B 0,C 180,E1 -27144.025,E2 -27144.025} C_VEL
LIN {X 0,Y 121.663,Z 333.262,A -85,B 0,C 180,E1 -27145.486,E2 -27145.486} C_VEL
LIN {X 0,Y 120.882,Z 326.89,A -85,B 0,C 180,E1 -27149.741,E2 -27149.741} C_VEL
LIN {X 0,Y 119.872,Z 321.239,A -85,B 0,C 180,E1 -27153.914,E2 -27153.914} C_VEL
LIN {X 0,Y 118.935,Z 317.028,A -85,B 0,C 180,E1 -27157.413,E2 -27157.413} C_VEL
LIN {X 0,Y 118.04,Z 313.376,A -85,B 0,C 180,E1 -27160.885,E2 -27160.885} C_VEL
LIN {X 0,Y 116.491,Z 307.722,A -85,B 0,C 180,E1 -27167.81,E2 -27167.81} C_VEL
LIN {X 0,Y 115.314,Z 303.85,A -85,B 0,C 180,E1 -27176.506,E2 -27176.506} C_VEL
LIN {X 0,Y 115.449,Z 302.631,A -85,B 0,C 180,E1 -27180,E2 -27180} C_VEL
LIN {X 0,Y 115.867,Z 304.772,A -85,B 0,C 180,E1 -27190.485,E2 -27190.485} C_VEL
LIN {X 0,Y 116.587,Z 306.05,A -85,B 0,C 180,E1 -27193.953,E2 -27193.953} C_VEL
LIN {X 0,Y 118.274,Z 310.429,A -85,B 0,C 180,E1 -27200.887,E2 -27200.887} C_VEL
LIN {X 0,Y 119.355,Z 313.165,A -85,B 0,C 180,E1 -27204.342,E2 -27204.342} C_VEL
LIN {X 0,Y 120.977,Z 318.046,A -85,B 0,C 180,E1 -27209.376,E2 -27209.376} C_VEL
LIN {X 0,Y 122.379,Z 323.382,A -85,B 0,C 180,E1 -27214.056,E2 -27214.056} C_VEL
LIN {X 0,Y 123.108,Z 328.396,A -85,B 0,C 180,E1 -27217.859,E2 -27217.859} C_VEL
LIN {X 0,Y 122.956,Z 333.589,A -85,B 0,C 180,E1 -27221.255,E2 -27221.255} C_VEL
LIN {X 0,Y 122.568,Z 336.158,A -85,B 0,C 180,E1 -27222.827,E2 -27222.827} C_VEL
LIN {X 0,Y 121.502,Z 338.356,A -85,B 0,C 180,E1 -27223.812,E2 -27223.812} C_VEL
LIN {X 0,Y 118.63,Z 341.517,A -85,B 0,C 180,E1 -27224.655,E2 -27224.655} C_VEL
LIN {X 0,Y 111.28,Z 347.558,A -85,B 0,C 180,E1 -27225.843,E2 -27225.843} C_VEL
LIN {X 0,Y 108.695,Z 350.072,A -85,B 0,C 180,E1 -27226.908,E2 -27226.908} C_VEL
LIN {X 0,Y 102.396,Z 357.244,A -85,B 0,C 180,E1 -27231.849,E2 -27231.849} C_VEL
LIN {X 0,Y 97.095,Z 362.702,A -85,B 0,C 180,E1 -27237.12,E2 -27237.12} C_VEL
LIN {X 0,Y 92.612,Z 366.981,A -85,B 0,C 180,E1 -27242.914,E2 -27242.914} C_VEL
LIN {X 0,Y 90.16,Z 369.24,A -85,B 0,C 180,E1 -27247.06,E2 -27247.06} C_VEL
LIN {X 0,Y 88.187,Z 371.071,A -85,B 0,C 180,E1 -27251.41,E2 -27251.41} C_VEL
LIN {X 0,Y 85.774,Z 373.242,A -85,B 0,C 180,E1 -27259.496,E2 -27259.496} C_VEL
LIN {X 0,Y 84.885,Z 374.018,A -85,B 0,C 180,E1 -27265.25,E2 -27265.25} C_VEL
LIN {X 0,Y 84.662,Z 374.241,A -85,B 0,C 180,E1 -27269.999,E2 -27269.999} C_VEL
LIN {X 0,Y 84.885,Z 374.044,A -85,B 0,C 180,E1 -27274.749,E2 -27274.749} C_VEL
LIN {X 0,Y 85.633,Z 373.374,A -85,B 0,C 180,E1 -27279.982,E2 -27279.982} C_VEL
LIN {X 0,Y 88.145,Z 371.157,A -85,B 0,C 180,E1 -27288.598,E2 -27288.598} C_VEL
LIN {X 0,Y 91.314,Z 368.308,A -85,B 0,C 180,E1 -27295.043,E2 -27295.043} C_VEL
LIN {X 0,Y 95.442,Z 364.438,A -85,B 0,C 180,E1 -27301.028,E2 -27301.028} C_VEL
LIN {X 0,Y 100.499,Z 359.435,A -85,B 0,C 180,E1 -27306.47,E2 -27306.47} C_VEL
LIN {X 0,Y 106.269,Z 353.129,A -85,B 0,C 180,E1 -27311.402,E2 -27311.402} C_VEL
LIN {X 0,Y 112.748,Z 345.232,A -85,B 0,C 180,E1 -27315.794,E2 -27315.794} C_VEL
LIN {X 0,Y 115.907,Z 340.948,A -85,B 0,C 180,E1 -27317.683,E2 -27317.683} C_VEL
LIN {X 0,Y 116.737,Z 339.349,A -85,B 0,C 180,E1 -27318.529,E2 -27318.529} C_VEL
LIN {X 0,Y 117.62,Z 334.53,A -85,B 0,C 180,E1 -27321.787,E2 -27321.787} C_VEL
LIN {X 0,Y 117.573,Z 329.887,A -85,B 0,C 180,E1 -27325.4,E2 -27325.4} C_VEL
LIN {X 0,Y 116.896,Z 325.671,A -85,B 0,C 180,E1 -27329.224,E2 -27329.224} C_VEL
LIN {X 0,Y 116.14,Z 321.854,A -85,B 0,C 180,E1 -27333.009,E2 -27333.009} C_VEL
LIN {X 0,Y 114.8,Z 317.458,A -85,B 0,C 180,E1 -27338.449,E2 -27338.449} C_VEL
LIN {X 0,Y 114.104,Z 314.961,A -85,B 0,C 180,E1 -27342.063,E2 -27342.063} C_VEL
LIN {X 0,Y 112.946,Z 311.479,A -85,B 0,C 180,E1 -27349.241,E2 -27349.241} C_VEL
LIN {X 0,Y 112.389,Z 309.942,A -85,B 0,C 180,E1 -27356.415,E2 -27356.415} C_VEL
LIN {X 0,Y 112.557,Z 309.581,A -85,B 0,C 180,E1 -27360,E2 -27360} C_VEL
LIN {X 0,Y 112.581,Z 312.135,A -85,B 0,C 180,E1 -27367.172,E2 -27367.172} C_VEL
LIN {X 0,Y 113.113,Z 313.674,A -85,B 0,C 180,E1 -27370.742,E2 -27370.742} C_VEL
LIN {X 0,Y 114.179,Z 319.004,A -85,B 0,C 180,E1 -27377.924,E2 -27377.924} C_VEL
LIN {X 0,Y 114.929,Z 323.697,A -85,B 0,C 180,E1 -27382.607,E2 -27382.607} C_VEL
LIN {X 0,Y 115.802,Z 330.132,A -85,B 0,C 180,E1 -27388.057,E2 -27388.057} C_VEL
LIN {X 0,Y 116.218,Z 336.776,A -85,B 0,C 180,E1 -27392.974,E2 -27392.974} C_VEL
LIN {X 0,Y 116.191,Z 338.218,A -85,B 0,C 180,E1 -27393.942,E2 -27393.942} C_VEL
LIN {X 0,Y 113.516,Z 345.737,A -85,B 0,C 180,E1 -27397.686,E2 -27397.686} C_VEL
LIN {X 0,Y 109.529,Z 354.364,A -85,B 0,C 180,E1 -27402.447,E2 -27402.447} C_VEL
LIN {X 0,Y 106.796,Z 358.66,A -85,B 0,C 180,E1 -27404.974,E2 -27404.974} C_VEL
LIN {X 0,Y 100.601,Z 365.881,A -85,B 0,C 180,E1 -27409.744,E2 -27409.744} C_VEL
LIN {X 0,Y 96.176,Z 370.777,A -85,B 0,C 180,E1 -27414.226,E2 -27414.226} C_VEL
LIN {X 0,Y 91.587,Z 375.54,A -85,B 0,C 180,E1 -27420.081,E2 -27420.081} C_VEL
LIN {X 0,Y 87.931,Z 379.188,A -85,B 0,C 180,E1 -27426.445,E2 -27426.445} C_VEL
LIN {X 0,Y 86.224,Z 381.082,A -85,B 0,C 180,E1 -27430.972,E2 -27430.972} C_VEL
LIN {X 0,Y 84.364,Z 383.545,A -85,B 0,C 180,E1 -27440.41,E2 -27440.41} C_VEL
LIN {X 0,Y 84.151,Z 384.184,A -85,B 0,C 180,E1 -27445.21,E2 -27445.21} C_VEL
LIN {X 0,Y 84.336,Z 384.42,A -85,B 0,C 180,E1 -27450.001,E2 -27450.001} C_VEL
LIN {X 0,Y 84.151,Z 384.168,A -85,B 0,C 180,E1 -27454.791,E2 -27454.791} C_VEL
LIN {X 0,Y 84.364,Z 383.519,A -85,B 0,C 180,E1 -27459.592,E2 -27459.592} C_VEL
LIN {X 0,Y 86.224,Z 381.03,A -85,B 0,C 180,E1 -27469.029,E2 -27469.029} C_VEL
LIN {X 0,Y 89.038,Z 378.027,A -85,B 0,C 180,E1 -27475.731,E2 -27475.731} C_VEL
LIN {X 0,Y 92.988,Z 373.987,A -85,B 0,C 180,E1 -27481.943,E2 -27481.943} C_VEL
LIN {X 0,Y 98.581,Z 367.982,A -85,B 0,C 180,E1 -27488.352,E2 -27488.352} C_VEL
LIN {X 0,Y 104.648,Z 361.052,A -85,B 0,C 180,E1 -27493.502,E2 -27493.502} C_VEL
LIN {X 0,Y 107.774,Z 357.091,A -85,B 0,C 180,E1 -27495.834,E2 -27495.834} C_VEL
LIN {X 0,Y 111.068,Z 350.977,A -85,B 0,C 180,E1 -27499.405,E2 -27499.405} C_VEL
LIN {X 0,Y 114.762,Z 342.24,A -85,B 0,C 180,E1 -27503.937,E2 -27503.937} C_VEL
LIN {X 0,Y 116.163,Z 337.886,A -85,B 0,C 180,E1 -27506.089,E2 -27506.089} C_VEL
LIN {X 0,Y 115.809,Z 331.159,A -85,B 0,C 180,E1 -27510.955,E2 -27510.955} C_VEL
LIN {X 0,Y 115.264,Z 326.434,A -85,B 0,C 180,E1 -27514.735,E2 -27514.735} C_VEL
LIN {X 0,Y 114.643,Z 322.308,A -85,B 0,C 180,E1 -27518.419,E2 -27518.419} C_VEL
LIN {X 0,Y 114.047,Z 318.751,A -85,B 0,C 180,E1 -27522.054,E2 -27522.054} C_VEL
LIN {X 0,Y 113.171,Z 314.566,A -85,B 0,C 180,E1 -27527.447,E2 -27527.447} C_VEL
LIN {X 0,Y 112.943,Z 313.447,A -85,B 0,C 180,E1 -27529.241,E2 -27529.241} C_VEL
LIN {X 0,Y 112.45,Z 309.168,A -85,B 0,C 180,E1 -27540,E2 -27540} C_VEL
LIN {X 0,Y 112.324,Z 310.486,A -85,B 0,C 180,E1 -27547.581,E2 -27547.581} C_VEL
LIN {X 0,Y 112.735,Z 311.272,A -85,B 0,C 180,E1 -27550.779,E2 -27550.779} C_VEL
LIN {X 0,Y 113.205,Z 312.803,A -85,B 0,C 180,E1 -27554.379,E2 -27554.379} C_VEL
LIN {X 0,Y 114.276,Z 315.87,A -85,B 0,C 180,E1 -27559.771,E2 -27559.771} C_VEL
LIN {X 0,Y 115.486,Z 320.086,A -85,B 0,C 180,E1 -27565.214,E2 -27565.214} C_VEL
LIN {X 0,Y 116.371,Z 323.458,A -85,B 0,C 180,E1 -27568.891,E2 -27568.891} C_VEL
LIN {X 0,Y 117.21,Z 327.656,A -85,B 0,C 180,E1 -27572.916,E2 -27572.916} C_VEL
LIN {X 0,Y 117.609,Z 332.811,A -85,B 0,C 180,E1 -27577.198,E2 -27577.198} C_VEL
LIN {X 0,Y 117.214,Z 336.605,A -85,B 0,C 180,E1 -27579.887,E2 -27579.887} C_VEL
LIN {X 0,Y 116.711,Z 339.015,A -85,B 0,C 180,E1 -27581.483,E2 -27581.483} C_VEL
LIN {X 0,Y 115.946,Z 340.627,A -85,B 0,C 180,E1 -27582.365,E2 -27582.365} C_VEL
LIN {X 0,Y 109.486,Z 349.099,A -85,B 0,C 180,E1 -27586.365,E2 -27586.365} C_VEL
LIN {X 0,Y 108.695,Z 350.072,A -85,B 0,C 180,E1 -27586.908,E2 -27586.908} C_VEL
LIN {X 0,Y 105.344,Z 353.517,A -85,B 0,C 180,E1 -27588.755,E2 -27588.755} C_VEL
LIN {X 0,Y 98.509,Z 358.689,A -85,B 0,C 180,E1 -27591.572,E2 -27591.572} C_VEL
LIN {X 0,Y 91.72,Z 363.161,A -85,B 0,C 180,E1 -27595.001,E2 -27595.001} C_VEL
LIN {X 0,Y 88.579,Z 365.509,A -85,B 0,C 180,E1 -27597.813,E2 -27597.813} C_VEL
LIN {X 0,Y 83.685,Z 369.668,A -85,B 0,C 180,E1 -27605.17,E2 -27605.17} C_VEL
LIN {X 0,Y 81.507,Z 371.498,A -85,B 0,C 180,E1 -27609.823,E2 -27609.823} C_VEL
LIN {X 0,Y 79.817,Z 372.869,A -85,B 0,C 180,E1 -27614.682,E2 -27614.682} C_VEL
LIN {X 0,Y 77.823,Z 374.445,A -85,B 0,C 180,E1 -27624.818,E2 -27624.818} C_VEL
LIN {X 0,Y 77.577,Z 374.668,A -85,B 0,C 180,E1 -27629.999,E2 -27629.999} C_VEL
LIN {X 0,Y 77.823,Z 374.47,A -85,B 0,C 180,E1 -27635.181,E2 -27635.181} C_VEL
LIN {X 0,Y 78.576,Z 373.887,A -85,B 0,C 180,E1 -27640.304,E2 -27640.304} C_VEL
LIN {X 0,Y 81.462,Z 371.583,A -85,B 0,C 180,E1 -27650.187,E2 -27650.187} C_VEL
LIN {X 0,Y 84.949,Z 368.733,A -85,B 0,C 180,E1 -27657.066,E2 -27657.066} C_VEL
LIN {X 0,Y 89.453,Z 364.863,A -85,B 0,C 180,E1 -27663.364,E2 -27663.364} C_VEL
LIN {X 0,Y 94.902,Z 359.86,A -85,B 0,C 180,E1 -27669.011,E2 -27669.011} C_VEL
LIN {X 0,Y 101.066,Z 353.554,A -85,B 0,C 180,E1 -27674.058,E2 -27674.058} C_VEL
LIN {X 0,Y 107.937,Z 345.655,A -85,B 0,C 180,E1 -27678.485,E2 -27678.485} C_VEL
LIN {X 0,Y 110.34,Z 342.627,A -85,B 0,C 180,E1 -27679.847,E2 -27679.847} C_VEL
LIN {X 0,Y 111.214,Z 340.96,A -85,B 0,C 180,E1 -27680.807,E2 -27680.807} C_VEL
LIN {X 0,Y 112.002,Z 337.498,A -85,B 0,C 180,E1 -27683.41,E2 -27683.41} C_VEL
LIN {X 0,Y 112.147,Z 333.676,A -85,B 0,C 180,E1 -27686.755,E2 -27686.755} C_VEL
LIN {X 0,Y 111.642,Z 328.76,A -85,B 0,C 180,E1 -27691.801,E2 -27691.801} C_VEL
LIN {X 0,Y 111.425,Z 326.916,A -85,B 0,C 180,E1 -27693.799,E2 -27693.799} C_VEL
LIN {X 0,Y 110.457,Z 322.717,A -85,B 0,C 180,E1 -27699.516,E2 -27699.516} C_VEL
LIN {X 0,Y 109.72,Z 319.459,A -85,B 0,C 180,E1 -27705.154,E2 -27705.154} C_VEL
LIN {X 0,Y 109.351,Z 317.863,A -85,B 0,C 180,E1 -27708.883,E2 -27708.883} C_VEL
LIN {X 0,Y 109.083,Z 316.861,A -85,B 0,C 180,E1 -27712.596,E2 -27712.596} C_VEL
LIN {X 0,Y 109.015,Z 316.224,A -85,B 0,C 180,E1 -27716.304,E2 -27716.304} C_VEL
LIN {X 0,Y 109.185,Z 315.928,A -85,B 0,C 180,E1 -27720,E2 -27720} C_VEL
LIN {X 0,Y 109.096,Z 318.515,A -85,B 0,C 180,E1 -27727.402,E2 -27727.402} C_VEL
LIN {X 0,Y 109.431,Z 320.24,A -85,B 0,C 180,E1 -27731.108,E2 -27731.108} C_VEL
LIN {X 0,Y 109.961,Z 324.962,A -85,B 0,C 180,E1 -27737.527,E2 -27737.527} C_VEL
LIN {X 0,Y 110.333,Z 328.616,A -85,B 0,C 180,E1 -27741.485,E2 -27741.485} C_VEL
LIN {X 0,Y 110.701,Z 334.94,A -85,B 0,C 180,E1 -27747.276,E2 -27747.276} C_VEL
LIN {X 0,Y 110.686,Z 340.085,A -85,B 0,C 180,E1 -27751.439,E2 -27751.439} C_VEL
LIN {X 0,Y 110.492,Z 341.472,A -85,B 0,C 180,E1 -27752.423,E2 -27752.423} C_VEL
LIN {X 0,Y 106.994,Z 349.327,A -85,B 0,C 180,E1 -27756.663,E2 -27756.663} C_VEL
LIN {X 0,Y 103.736,Z 355.44,A -85,B 0,C 180,E1 -27760.344,E2 -27760.344} C_VEL
LIN {X 0,Y 101.843,Z 358.229,A -85,B 0,C 180,E1 -27762.112,E2 -27762.112} C_VEL
LIN {X 0,Y 95.267,Z 365.453,A -85,B 0,C 180,E1 -27766.97,E2 -27766.97} C_VEL
LIN {X 0,Y 90.432,Z 370.345,A -85,B 0,C 180,E1 -27771.558,E2 -27771.558} C_VEL
LIN {X 0,Y 85.478,Z 375.112,A -85,B 0,C 180,E1 -27777.695,E2 -27777.695} C_VEL
LIN {X 0,Y 81.435,Z 378.758,A -85,B 0,C 180,E1 -27784.437,E2 -27784.437} C_VEL
LIN {X 0,Y 79.519,Z 380.654,A -85,B 0,C 180,E1 -27789.298,E2 -27789.298} C_VEL
LIN {X 0,Y 77.346,Z 383.116,A -85,B 0,C 180,E1 -27799.53,E2 -27799.53} C_VEL
LIN {X 0,Y 77.067,Z 383.756,A -85,B 0,C 180,E1 -27804.768,E2 -27804.768} C_VEL
LIN {X 0,Y 77.247,Z 383.993,A -85,B 0,C 180,E1 -27810.001,E2 -27810.001} C_VEL
LIN {X 0,Y 77.067,Z 383.74,A -85,B 0,C 180,E1 -27815.233,E2 -27815.233} C_VEL
LIN {X 0,Y 77.346,Z 383.09,A -85,B 0,C 180,E1 -27820.471,E2 -27820.471} C_VEL
LIN {X 0,Y 79.519,Z 380.601,A -85,B 0,C 180,E1 -27830.704,E2 -27830.704} C_VEL
LIN {X 0,Y 82.673,Z 377.596,A -85,B 0,C 180,E1 -27837.877,E2 -27837.877} C_VEL
LIN {X 0,Y 87.015,Z 373.556,A -85,B 0,C 180,E1 -27844.429,E2 -27844.429} C_VEL
LIN {X 0,Y 92.514,Z 368.133,A -85,B 0,C 180,E1 -27850.565,E2 -27850.565} C_VEL
LIN {X 0,Y 99.588,Z 360.619,A -85,B 0,C 180,E1 -27856.333,E2 -27856.333} C_VEL
LIN {X 0,Y 102.776,Z 356.645,A -85,B 0,C 180,E1 -27858.782,E2 -27858.782} C_VEL
LIN {X 0,Y 106.227,Z 350.511,A -85,B 0,C 180,E1 -27862.555,E2 -27862.555} C_VEL
LIN {X 0,Y 110.107,Z 342.201,A -85,B 0,C 180,E1 -27867.042,E2 -27867.042} C_VEL
LIN {X 0,Y 110.533,Z 341.018,A -85,B 0,C 180,E1 -27867.679,E2 -27867.679} C_VEL
LIN {X 0,Y 110.633,Z 336.096,A -85,B 0,C 180,E1 -27871.549,E2 -27871.549} C_VEL
LIN {X 0,Y 110.34,Z 330.307,A -85,B 0,C 180,E1 -27876.663,E2 -27876.663} C_VEL
LIN {X 0,Y 110.15,Z 327.397,A -85,B 0,C 180,E1 -27879.457,E2 -27879.457} C_VEL
LIN {X 0,Y 109.719,Z 323.513,A -85,B 0,C 180,E1 -27883.911,E2 -27883.911} C_VEL
LIN {X 0,Y 109.314,Z 319.961,A -85,B 0,C 180,E1 -27888.879,E2 -27888.879} C_VEL
LIN {X 0,Y 108.845,Z 316.82,A -85,B 0,C 180,E1 -27896.298,E2 -27896.298} C_VEL
LIN {X 0,Y 109.084,Z 315.553,A -85,B 0,C 180,E1 -27900,E2 -27900} C_VEL
LIN {X 0,Y 108.875,Z 316.678,A -85,B 0,C 180,E1 -27907.418,E2 -27907.418} C_VEL
LIN {X 0,Y 109.166,Z 317.637,A -85,B 0,C 180,E1 -27911.136,E2 -27911.136} C_VEL
LIN {X 0,Y 109.668,Z 319.82,A -85,B 0,C 180,E1 -27915.996,E2 -27915.996} C_VEL
LIN {X 0,Y 110.326,Z 322.418,A -85,B 0,C 180,E1 -27920.51,E2 -27920.51} C_VEL
LIN {X 0,Y 111.256,Z 326.697,A -85,B 0,C 180,E1 -27926.244,E2 -27926.244} C_VEL
LIN {X 0,Y 111.946,Z 331.718,A -85,B 0,C 180,E1 -27931.64,E2 -27931.64} C_VEL
LIN {X 0,Y 112.08,Z 335.757,A -85,B 0,C 180,E1 -27935.395,E2 -27935.395} C_VEL
LIN {X 0,Y 111.589,Z 339.078,A -85,B 0,C 180,E1 -27938.042,E2 -27938.042} C_VEL
LIN {X 0,Y 111.21,Z 340.622,A -85,B 0,C 180,E1 -27939.195,E2 -27939.195} C_VEL
LIN {X 0,Y 110.381,Z 342.279,A -85,B 0,C 180,E1 -27940.176,E2 -27940.176} C_VEL
LIN {X 0,Y 103.342,Z 350.847,A -85,B 0,C 180,E1 -27944.431,E2 -27944.431} C_VEL
LIN {X 0,Y 96.918,Z 357.673,A -85,B 0,C 180,E1 -27949.258,E2 -27949.258} C_VEL
LIN {X 0,Y 91.235,Z 363.13,A -85,B 0,C 180,E1 -27954.707,E2 -27954.707} C_VEL
LIN {X 0,Y 88.579,Z 365.509,A -85,B 0,C 180,E1 -27957.813,E2 -27957.813} C_VEL
LIN {X 0,Y 85.608,Z 367.639,A -85,B 0,C 180,E1 -27960.877,E2 -27960.877} C_VEL
LIN {X 0,Y 79.577,Z 370.632,A -85,B 0,C 180,E1 -27965.936,E2 -27965.936} C_VEL
LIN {X 0,Y 75.035,Z 372.508,A -85,B 0,C 180,E1 -27970.581,E2 -27970.581} C_VEL
LIN {X 0,Y 72.643,Z 373.593,A -85,B 0,C 180,E1 -27974.706,E2 -27974.706} C_VEL
LIN {X 0,Y 72.17,Z 373.834,A -85,B 0,C 180,E1 -27976.205,E2 -27976.205} C_VEL
LIN {X 0,Y 70.767,Z 374.872,A -85,B 0,C 180,E1 -27984.3,E2 -27984.3} C_VEL
LIN {X 0,Y 70.491,Z 375.094,A -85,B 0,C 180,E1 -27989.999,E2 -27989.999} C_VEL
LIN {X 0,Y 71.635,Z 374.312,A -85,B 0,C 180,E1 -28001.315,E2 -28001.315} C_VEL
LIN {X 0,Y 74.85,Z 372.009,A -85,B 0,C 180,E1 -28012.059,E2 -28012.059} C_VEL
LIN {X 0,Y 78.714,Z 369.159,A -85,B 0,C 180,E1 -28019.41,E2 -28019.41} C_VEL
LIN {X 0,Y 83.635,Z 365.288,A -85,B 0,C 180,E1 -28026.03,E2 -28026.03} C_VEL
LIN {X 0,Y 89.493,Z 360.286,A -85,B 0,C 180,E1 -28031.875,E2 -28031.875} C_VEL
LIN {X 0,Y 96.105,Z 353.978,A -85,B 0,C 180,E1 -28036.994,E2 -28036.994} C_VEL
LIN {X 0,Y 103.386,Z 346.078,A -85,B 0,C 180,E1 -28041.42,E2 -28041.42} C_VEL
LIN {X 0,Y 105.053,Z 344.138,A -85,B 0,C 180,E1 -28042.31,E2 -28042.31} C_VEL
LIN {X 0,Y 105.838,Z 342.617,A -85,B 0,C 180,E1 -28043.299,E2 -28043.299} C_VEL
LIN {X 0,Y 106.652,Z 338.443,A -85,B 0,C 180,E1 -28047.067,E2 -28047.067} C_VEL
LIN {X 0,Y 106.575,Z 333.579,A -85,B 0,C 180,E1 -28052.509,E2 -28052.509} C_VEL
LIN {X 0,Y 106.524,Z 331.812,A -85,B 0,C 180,E1 -28054.606,E2 -28054.606} C_VEL
LIN {X 0,Y 105.941,Z 327.799,A -85,B 0,C 180,E1 -28060.628,E2 -28060.628} C_VEL
LIN {X 0,Y 105.672,Z 325.652,A -85,B 0,C 180,E1 -28064.572,E2 -28064.572} C_VEL
LIN {X 0,Y 105.411,Z 324.046,A -85,B 0,C 180,E1 -28068.462,E2 -28068.462} C_VEL
LIN {X 0,Y 105.26,Z 322.942,A -85,B 0,C 180,E1 -28072.326,E2 -28072.326} C_VEL
LIN {X 0,Y 105.432,Z 322.057,A -85,B 0,C 180,E1 -28079.141,E2 -28079.141} C_VEL
LIN {X 0,Y 105.421,Z 322.187,A -85,B 0,C 180,E1 -28080.332,E2 -28080.332} C_VEL
LIN {X 0,Y 105.205,Z 324.698,A -85,B 0,C 180,E1 -28087.678,E2 -28087.678} C_VEL
LIN {X 0,Y 105.398,Z 327.934,A -85,B 0,C 180,E1 -28093.496,E2 -28093.496} C_VEL
LIN {X 0,Y 105.493,Z 329.255,A -85,B 0,C 180,E1 -28095.455,E2 -28095.455} C_VEL
LIN {X 0,Y 105.56,Z 332.531,A -85,B 0,C 180,E1 -28099.444,E2 -28099.444} C_VEL
LIN {X 0,Y 105.442,Z 338.701,A -85,B 0,C 180,E1 -28105.673,E2 -28105.673} C_VEL
LIN {X 0,Y 105.148,Z 343.142,A -85,B 0,C 180,E1 -28109.668,E2 -28109.668} C_VEL
LIN {X 0,Y 104.55,Z 344.978,A -85,B 0,C 180,E1 -28110.954,E2 -28110.954} C_VEL
LIN {X 0,Y 100.838,Z 351.918,A -85,B 0,C 180,E1 -28115.023,E2 -28115.023} C_VEL
LIN {X 0,Y 97.072,Z 357.789,A -85,B 0,C 180,E1 -28118.895,E2 -28118.895} C_VEL
LIN {X 0,Y 92.432,Z 362.773,A -85,B 0,C 180,E1 -28122.156,E2 -28122.156} C_VEL
LIN {X 0,Y 84.916,Z 369.914,A -85,B 0,C 180,E1 -28128.54,E2 -28128.54} C_VEL
LIN {X 0,Y 79.516,Z 374.682,A -85,B 0,C 180,E1 -28134.936,E2 -28134.936} C_VEL
LIN {X 0,Y 75.063,Z 378.33,A -85,B 0,C 180,E1 -28142.087,E2 -28142.087} C_VEL
LIN {X 0,Y 72.882,Z 380.224,A -85,B 0,C 180,E1 -28147.312,E2 -28147.312} C_VEL
LIN {X 0,Y 70.346,Z 382.687,A -85,B 0,C 180,E1 -28158.475,E2 -28158.475} C_VEL
LIN {X 0,Y 69.988,Z 383.328,A -85,B 0,C 180,E1 -28164.238,E2 -28164.238} C_VEL
LIN {X 0,Y 70.16,Z 383.566,A -85,B 0,C 180,E1 -28170.001,E2 -28170.001} C_VEL
LIN {X 0,Y 69.988,Z 383.311,A -85,B 0,C 180,E1 -28175.764,E2 -28175.764} C_VEL
LIN {X 0,Y 70.346,Z 382.66,A -85,B 0,C 180,E1 -28181.527,E2 -28181.527} C_VEL
LIN {X 0,Y 72.882,Z 380.17,A -85,B 0,C 180,E1 -28192.689,E2 -28192.689} C_VEL
LIN {X 0,Y 76.446,Z 377.166,A -85,B 0,C 180,E1 -28200.375,E2 -28200.375} C_VEL
LIN {X 0,Y 81.232,Z 373.126,A -85,B 0,C 180,E1 -28207.275,E2 -28207.275} C_VEL
LIN {X 0,Y 87.835,Z 367.105,A -85,B 0,C 180,E1 -28214.161,E2 -28214.161} C_VEL
LIN {X 0,Y 94.794,Z 360.187,A -85,B 0,C 180,E1 -28219.46,E2 -28219.46} C_VEL
LIN {X 0,Y 97.051,Z 357.586,A -85,B 0,C 180,E1 -28221.122,E2 -28221.122} C_VEL
LIN {X 0,Y 100.796,Z 351.691,A -85,B 0,C 180,E1 -28225.013,E2 -28225.013} C_VEL
LIN {X 0,Y 104.55,Z 344.746,A -85,B 0,C 180,E1 -28229.011,E2 -28229.011} C_VEL
LIN {X 0,Y 105.071,Z 342.846,A -85,B 0,C 180,E1 -28230.407,E2 -28230.407} C_VEL
LIN {X 0,Y 105.36,Z 337.393,A -85,B 0,C 180,E1 -28235.361,E2 -28235.361} C_VEL
LIN {X 0,Y 105.457,Z 332.302,A -85,B 0,C 180,E1 -28240.536,E2 -28240.536} C_VEL
LIN {X 0,Y 105.362,Z 329.052,A -85,B 0,C 180,E1 -28244.525,E2 -28244.525} C_VEL
LIN {X 0,Y 105.216,Z 326.421,A -85,B 0,C 180,E1 -28248.441,E2 -28248.441} C_VEL
LIN {X 0,Y 105.079,Z 324.447,A -85,B 0,C 180,E1 -28252.313,E2 -28252.313} C_VEL
LIN {X 0,Y 105.368,Z 321.748,A -85,B 0,C 180,E1 -28260,E2 -28260} C_VEL
LIN {X 0,Y 105.125,Z 322.054,A -85,B 0,C 180,E1 -28263.833,E2 -28263.833} C_VEL
LIN {X 0,Y 105.236,Z 323.826,A -85,B 0,C 180,E1 -28271.558,E2 -28271.558} C_VEL
LIN {X 0,Y 105.567,Z 326.032,A -85,B 0,C 180,E1 -28276.635,E2 -28276.635} C_VEL
LIN {X 0,Y 106.039,Z 329.124,A -85,B 0,C 180,E1 -28281.89,E2 -28281.89} C_VEL
LIN {X 0,Y 106.352,Z 331.617,A -85,B 0,C 180,E1 -28285.438,E2 -28285.438} C_VEL
LIN {X 0,Y 106.607,Z 336.363,A -85,B 0,C 180,E1 -28291.015,E2 -28291.015} C_VEL
LIN {X 0,Y 106.482,Z 339.36,A -85,B 0,C 180,E1 -28294.127,E2 -28294.127} C_VEL
